KUKA KRL program: PickPlaceTrayTeach.src, PickPlaceTrayTeach.dat

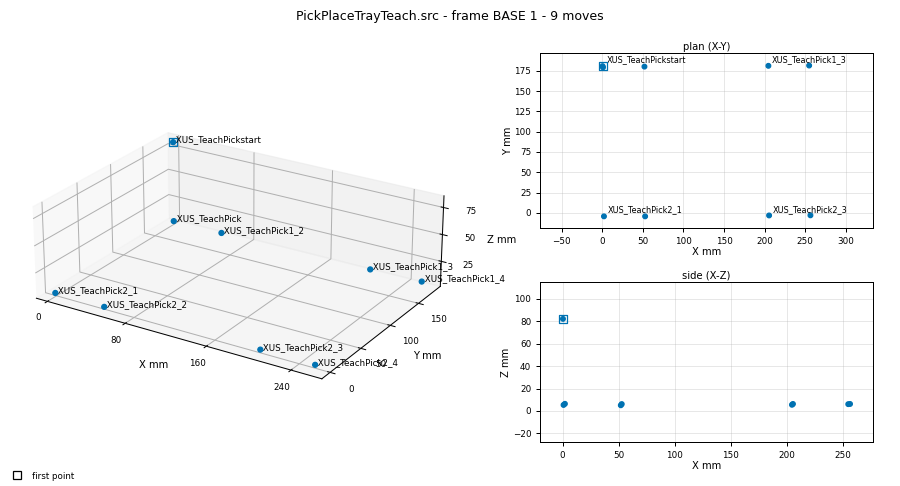
[picture p0: tool path of PickPlaceTrayTeach.src in frame BASE 1, 9 of 139 moves have a stored position in this frame; points joined in program order, loops and branches not executed]
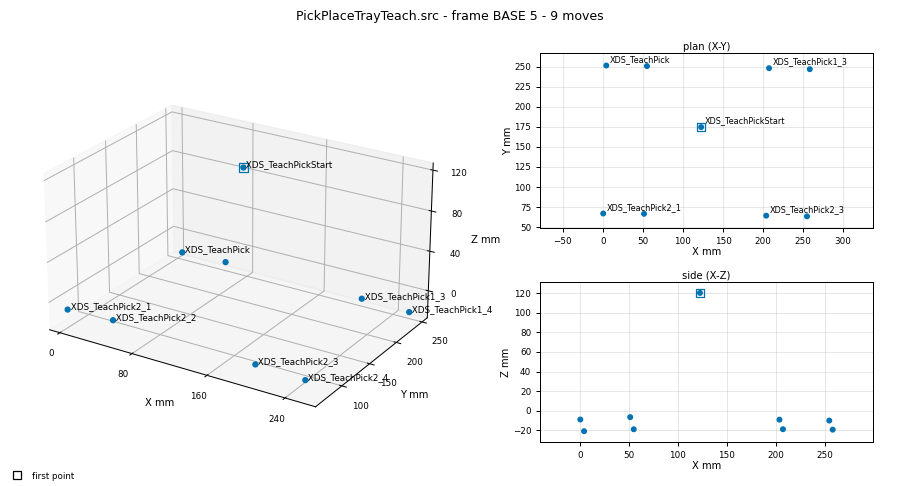
[picture p1: tool path of PickPlaceTrayTeach.src in frame BASE 5, 9 of 139 moves have a stored position in this frame; points joined in program order, loops and branches not executed]
--- PickPlaceTrayTeach.src ---
&ACCESS RVO1
&REL 58
&PARAM DISKPATH = KRC:\R1\Program
DEF PickPlaceTrayTeach()

   ;FOLD INI;%{PE}
      ;FOLD BASISTECH INI
         GLOBAL INTERRUPT DECL 3 WHEN $STOPMESS == TRUE DO IR_STOPM()
         INTERRUPT ON 3
         BAS(#INITMOV, 0)
      ;ENDFOLD (BASISTECH INI)
      ;FOLD USER INI
         ;Make your modifications here
      ;ENDFOLD (USER INI)
      ;ENDFOLD (INI)

            US_Pick[1,1]= XUS_TeachPick
            US_Pick[1,2]= XUS_TeachPick1_2
            US_Pick[1,3]= XUS_TeachPick1_3
            US_Pick[1,4]= XUS_TeachPick1_4
            US_Pick[2,1]= XUS_TeachPick2_1
            US_Pick[2,2]= XUS_TeachPick2_2
            US_Pick[2,3]= XUS_TeachPick2_3
            US_Pick[2,4]= XUS_TeachPick2_4



            DS_Pick[1,1]= XDS_TeachPick
            DS_Pick[1,2]= XDS_TeachPick1_2
            DS_Pick[1,3]= XDS_TeachPick1_3
            DS_Pick[1,4]= XDS_TeachPick1_4
            DS_Pick[2,1]= XDS_TeachPick2_1
            DS_Pick[2,2]= XDS_TeachPick2_2
            DS_Pick[2,3]= XDS_TeachPick2_3
            DS_Pick[2,4]= XDS_TeachPick2_4




            GOTO EndOfModule


        RtoIMM_SeqNumber=1





;move joint 1 to turn robot towards upstacker from home
   ;FOLD SPTP US_A1Turn Vel=100 % PDAT3 Tool[0] Base[0] ;%{PE}
      ;FOLD Parameters ;%{h}
         ;Params IlfProvider=kukaroboter.basistech.inlineforms.movement.spline; Kuka.IsGlobalPoint=False; Kuka.PointName=US_A1Turn; Kuka.BlendingEnabled=False; Kuka.MoveDataPtpName=PDAT3; Kuka.VelocityPtp=100; Kuka.VelocityFieldEnabled=True; Kuka.ColDetectFieldEnabled=True; Kuka.CurrentCDSetIndex=0; Kuka.MovementParameterFieldEnabled=True; IlfCommand=SPTP
      ;ENDFOLD
      SPTP XUS_A1Turn WITH $VEL_AXIS[1] = SVEL_JOINT(100.0), $TOOL = STOOL2(FUS_A1Turn), $BASE = SBASE(FUS_A1Turn.BASE_NO), $IPO_MODE = SIPO_MODE(FUS_A1Turn.IPO_FRAME), $LOAD = SLOAD(FUS_A1Turn.TOOL_NO), $ACC_AXIS[1] = SACC_JOINT(PPDAT3), $APO = SAPO_PTP(PPDAT3), $GEAR_JERK[1] = SGEAR_JERK(PPDAT3), $COLLMON_TOL_PRO[1] = USE_CM_PRO_VALUES(0)
      ;ENDFOLD



;FOLD SPTP US_TeachPickstart Vel=100 % PDAT8 Tool[1]:BlankPick Base[1]:UpStacker ;%{PE}
;FOLD Parameters ;%{h}
;Params IlfProvider=kukaroboter.basistech.inlineforms.movement.spline; Kuka.IsGlobalPoint=False; Kuka.PointName=US_TeachPickstart; Kuka.BlendingEnabled=False; Kuka.MoveDataPtpName=PDAT8; Kuka.VelocityPtp=100; Kuka.VelocityFieldEnabled=True; Kuka.ColDetectFieldEnabled=True; Kuka.CurrentCDSetIndex=0; Kuka.MovementParameterFieldEnabled=True; IlfCommand=SPTP
;ENDFOLD
SPTP XUS_TeachPickstart WITH $VEL_AXIS[1] = SVEL_JOINT(100.0), $TOOL = STOOL2(FUS_TeachPickstart), $BASE = SBASE(FUS_TeachPickstart.BASE_NO), $IPO_MODE = SIPO_MODE(FUS_TeachPickstart.IPO_FRAME), $LOAD = SLOAD(FUS_TeachPickstart.TOOL_NO), $ACC_AXIS[1] = SACC_JOINT(PPDAT8), $APO = SAPO_PTP(PPDAT8), $GEAR_JERK[1] = SGEAR_JERK(PPDAT8), $COLLMON_TOL_PRO[1] = USE_CM_PRO_VALUES(0)
;ENDFOLD

 US_PickApproach[1,1] = US_Pick[1,1]
 US_PickApproach[1,1].Z = US_PickApproach[1,1].Z + 100
 US_PickApproachSlow[1,1].Z = US_PickApproach[1,1].Z - 65
 SLIN US_PickApproach[1,1] with $TOOL=TOOL_DATA[1],$BASE=BASE_DATA[1],$LOAD=LOAD_DATA[1],$VEL.CP = 2
 SLIN US_PickApproachSlow[1,1] with $TOOL=TOOL_DATA[1],$BASE=BASE_DATA[1],$LOAD=LOAD_DATA[1],$VEL.CP = 2
;FOLD SLIN US_TeachPick Vel=1 m/s CPDAT15 Tool[1]:BlankPick Base[1]:UpStacker ;%{PE}
;FOLD Parameters ;%{h}
;Params IlfProvider=kukaroboter.basistech.inlineforms.movement.spline; Kuka.IsGlobalPoint=False; Kuka.PointName=US_TeachPick; Kuka.BlendingEnabled=False; Kuka.MoveDataName=CPDAT15; Kuka.VelocityPath=1; Kuka.VelocityFieldEnabled=True; Kuka.ColDetectFieldEnabled=True; Kuka.CurrentCDSetIndex=0; Kuka.MovementParameterFieldEnabled=True; IlfCommand=SLIN
;ENDFOLD
SLIN XUS_TeachPick WITH $VEL = SVEL_CP(1.0, , LCPDAT15), $TOOL = STOOL2(FUS_TeachPick), $BASE = SBASE(FUS_TeachPick.BASE_NO), $IPO_MODE = SIPO_MODE(FUS_TeachPick.IPO_FRAME), $LOAD = SLOAD(FUS_TeachPick.TOOL_NO), $ACC = SACC_CP(LCPDAT15), $ORI_TYPE = SORI_TYP(LCPDAT15), $APO = SAPO(LCPDAT15), $JERK = SJERK(LCPDAT15), $COLLMON_TOL_PRO[1] = USE_CM_PRO_VALUES(0)
;ENDFOLD
US_Pick[1,1]= XUS_TeachPick
SLIN US_Pick[1,1] with $TOOL=TOOL_DATA[1],$BASE=BASE_DATA[1],$LOAD=LOAD_DATA[1],$VEL.CP = 0.1
SLIN US_PickApproach[1,1] with $TOOL=TOOL_DATA[1],$BASE=BASE_DATA[1],$LOAD=LOAD_DATA[1],$VEL.CP = 2

US_PickApproach[1,2] = US_Pick[1,2]
 US_PickApproach[1,2].Z = US_PickApproach[1,2].Z + 100
 US_PickApproachSlow[1,2].Z = US_PickApproach[1,2].Z - 65
 SLIN US_PickApproach[1,2] with $TOOL=TOOL_DATA[1],$BASE=BASE_DATA[1],$LOAD=LOAD_DATA[1],$VEL.CP = 2
 SLIN US_PickApproachSlow[1,2] with $TOOL=TOOL_DATA[1],$BASE=BASE_DATA[1],$LOAD=LOAD_DATA[1],$VEL.CP = 2
;FOLD SLIN US_TeachPick1_2 Vel=1 m/s CPDAT07 Tool[1]:BlankPick Base[1]:UpStacker ;%{PE}
;FOLD Parameters ;%{h}
;Params IlfProvider=kukaroboter.basistech.inlineforms.movement.spline; Kuka.IsGlobalPoint=False; Kuka.PointName=US_TeachPick1_2; Kuka.BlendingEnabled=False; Kuka.MoveDataName=CPDAT07; Kuka.VelocityPath=1; Kuka.VelocityFieldEnabled=True; Kuka.ColDetectFieldEnabled=True; Kuka.CurrentCDSetIndex=0; Kuka.MovementParameterFieldEnabled=True; IlfCommand=SLIN
;ENDFOLD
SLIN XUS_TeachPick1_2 WITH $VEL = SVEL_CP(1.0, , LCPDAT07), $TOOL = STOOL2(FUS_TeachPick1_2), $BASE = SBASE(FUS_TeachPick1_2.BASE_NO), $IPO_MODE = SIPO_MODE(FUS_TeachPick1_2.IPO_FRAME), $LOAD = SLOAD(FUS_TeachPick1_2.TOOL_NO), $ACC = SACC_CP(LCPDAT07), $ORI_TYPE = SORI_TYP(LCPDAT07), $APO = SAPO(LCPDAT07), $JERK = SJERK(LCPDAT07), $COLLMON_TOL_PRO[1] = USE_CM_PRO_VALUES(0)
;ENDFOLD
US_Pick[1,2]= XUS_TeachPick
SLIN US_Pick[1,2] with $TOOL=TOOL_DATA[1],$BASE=BASE_DATA[1],$LOAD=LOAD_DATA[1],$VEL.CP = 0.1
 SLIN US_PickApproach[1,2] with $TOOL=TOOL_DATA[1],$BASE=BASE_DATA[1],$LOAD=LOAD_DATA[1],$VEL.CP = 2

US_PickApproach[1,3] = US_Pick[1,3]
 US_PickApproach[1,3].Z = US_PickApproach[1,3].Z + 100
 US_PickApproachSlow[1,3].Z = US_PickApproach[1,3].Z - 65
 SLIN US_PickApproach[1,3] with $TOOL=TOOL_DATA[1],$BASE=BASE_DATA[1],$LOAD=LOAD_DATA[1],$VEL.CP = 2
 SLIN US_PickApproachSlow[1,3] with $TOOL=TOOL_DATA[1],$BASE=BASE_DATA[1],$LOAD=LOAD_DATA[1],$VEL.CP = 2
;FOLD SLIN US_TeachPick1_3 Vel=1 m/s CPDAT08 Tool[1]:BlankPick Base[1]:UpStacker ;%{PE}
;FOLD Parameters ;%{h}
;Params IlfProvider=kukaroboter.basistech.inlineforms.movement.spline; Kuka.IsGlobalPoint=False; Kuka.PointName=US_TeachPick1_3; Kuka.BlendingEnabled=False; Kuka.MoveDataName=CPDAT08; Kuka.VelocityPath=1; Kuka.VelocityFieldEnabled=True; Kuka.ColDetectFieldEnabled=True; Kuka.CurrentCDSetIndex=0; Kuka.MovementParameterFieldEnabled=True; IlfCommand=SLIN
;ENDFOLD
SLIN XUS_TeachPick1_3 WITH $VEL = SVEL_CP(1.0, , LCPDAT08), $TOOL = STOOL2(FUS_TeachPick1_3), $BASE = SBASE(FUS_TeachPick1_3.BASE_NO), $IPO_MODE = SIPO_MODE(FUS_TeachPick1_3.IPO_FRAME), $LOAD = SLOAD(FUS_TeachPick1_3.TOOL_NO), $ACC = SACC_CP(LCPDAT08), $ORI_TYPE = SORI_TYP(LCPDAT08), $APO = SAPO(LCPDAT08), $JERK = SJERK(LCPDAT08), $COLLMON_TOL_PRO[1] = USE_CM_PRO_VALUES(0)
;ENDFOLD
US_Pick[1,3]= XUS_TeachPick
SLIN US_Pick[1,3] with $TOOL=TOOL_DATA[1],$BASE=BASE_DATA[1],$LOAD=LOAD_DATA[1],$VEL.CP = 0.1
 SLIN US_PickApproach[1,3] with $TOOL=TOOL_DATA[1],$BASE=BASE_DATA[1],$LOAD=LOAD_DATA[1],$VEL.CP = 2

US_PickApproach[1,4] = US_Pick[1,4]
 US_PickApproach[1,4].Z = US_PickApproach[1,4].Z + 100
 US_PickApproachSlow[1,4].Z = US_PickApproach[1,4].Z - 65
 SLIN US_PickApproach[1,4] with $TOOL=TOOL_DATA[1],$BASE=BASE_DATA[1],$LOAD=LOAD_DATA[1],$VEL.CP = 2
 SLIN US_PickApproachSlow[1,4] with $TOOL=TOOL_DATA[1],$BASE=BASE_DATA[1],$LOAD=LOAD_DATA[1],$VEL.CP = 2
;FOLD SLIN US_TeachPick1_4 Vel=1 m/s CPDAT09 Tool[1]:BlankPick Base[1]:UpStacker ;%{PE}
;FOLD Parameters ;%{h}
;Params IlfProvider=kukaroboter.basistech.inlineforms.movement.spline; Kuka.IsGlobalPoint=False; Kuka.PointName=US_TeachPick1_4; Kuka.BlendingEnabled=False; Kuka.MoveDataName=CPDAT09; Kuka.VelocityPath=1; Kuka.VelocityFieldEnabled=True; Kuka.ColDetectFieldEnabled=True; Kuka.CurrentCDSetIndex=0; Kuka.MovementParameterFieldEnabled=True; IlfCommand=SLIN
;ENDFOLD
SLIN XUS_TeachPick1_4 WITH $VEL = SVEL_CP(1.0, , LCPDAT09), $TOOL = STOOL2(FUS_TeachPick1_4), $BASE = SBASE(FUS_TeachPick1_4.BASE_NO), $IPO_MODE = SIPO_MODE(FUS_TeachPick1_4.IPO_FRAME), $LOAD = SLOAD(FUS_TeachPick1_4.TOOL_NO), $ACC = SACC_CP(LCPDAT09), $ORI_TYPE = SORI_TYP(LCPDAT09), $APO = SAPO(LCPDAT09), $JERK = SJERK(LCPDAT09), $COLLMON_TOL_PRO[1] = USE_CM_PRO_VALUES(0)
;ENDFOLD
US_Pick[1,4]= XUS_TeachPick
SLIN US_Pick[1,4] with $TOOL=TOOL_DATA[1],$BASE=BASE_DATA[1],$LOAD=LOAD_DATA[1],$VEL.CP = 0.1
 SLIN US_PickApproach[1,4] with $TOOL=TOOL_DATA[1],$BASE=BASE_DATA[1],$LOAD=LOAD_DATA[1],$VEL.CP = 2

US_PickApproach[2,1] = US_Pick[2,1]
 US_PickApproach[2,1].Z = US_PickApproach[2,1].Z + 100
 US_PickApproachSlow[2,1].Z = US_PickApproach[2,1].Z - 65
 SLIN US_PickApproach[2,1] with $TOOL=TOOL_DATA[1],$BASE=BASE_DATA[1],$LOAD=LOAD_DATA[1],$VEL.CP = 2
 SLIN US_PickApproachSlow[2,1] with $TOOL=TOOL_DATA[1],$BASE=BASE_DATA[1],$LOAD=LOAD_DATA[1],$VEL.CP = 2
;FOLD SLIN US_TeachPick2_1 Vel=1 m/s CPDAT11 Tool[1]:BlankPick Base[1]:UpStacker ;%{PE}
;FOLD Parameters ;%{h}
;Params IlfProvider=kukaroboter.basistech.inlineforms.movement.spline; Kuka.IsGlobalPoint=False; Kuka.PointName=US_TeachPick2_1; Kuka.BlendingEnabled=False; Kuka.MoveDataName=CPDAT11; Kuka.VelocityPath=1; Kuka.VelocityFieldEnabled=True; Kuka.ColDetectFieldEnabled=True; Kuka.CurrentCDSetIndex=0; Kuka.MovementParameterFieldEnabled=True; IlfCommand=SLIN
;ENDFOLD
SLIN XUS_TeachPick2_1 WITH $VEL = SVEL_CP(1.0, , LCPDAT11), $TOOL = STOOL2(FUS_TeachPick2_1), $BASE = SBASE(FUS_TeachPick2_1.BASE_NO), $IPO_MODE = SIPO_MODE(FUS_TeachPick2_1.IPO_FRAME), $LOAD = SLOAD(FUS_TeachPick2_1.TOOL_NO), $ACC = SACC_CP(LCPDAT11), $ORI_TYPE = SORI_TYP(LCPDAT11), $APO = SAPO(LCPDAT11), $JERK = SJERK(LCPDAT11), $COLLMON_TOL_PRO[1] = USE_CM_PRO_VALUES(0)
;ENDFOLD
US_Pick[2,1]= XUS_TeachPick
SLIN US_Pick[2,1] with $TOOL=TOOL_DATA[1],$BASE=BASE_DATA[1],$LOAD=LOAD_DATA[1],$VEL.CP = 0.1
 SLIN US_PickApproach[2,1] with $TOOL=TOOL_DATA[1],$BASE=BASE_DATA[1],$LOAD=LOAD_DATA[1],$VEL.CP = 2

US_PickApproach[2,2] = US_Pick[2,2]
 US_PickApproach[2,2].Z = US_PickApproach[2,2].Z + 100
 US_PickApproachSlow[2,2].Z = US_PickApproach[2,2].Z - 65
 SLIN US_PickApproach[2,2] with $TOOL=TOOL_DATA[1],$BASE=BASE_DATA[1],$LOAD=LOAD_DATA[1],$VEL.CP = 2
 SLIN US_PickApproachSlow[2,2] with $TOOL=TOOL_DATA[1],$BASE=BASE_DATA[1],$LOAD=LOAD_DATA[1],$VEL.CP = 2
;FOLD SLIN US_TeachPick2_2 Vel=1 m/s CPDAT12 Tool[1]:BlankPick Base[1]:UpStacker ;%{PE}
;FOLD Parameters ;%{h}
;Params IlfProvider=kukaroboter.basistech.inlineforms.movement.spline; Kuka.IsGlobalPoint=False; Kuka.PointName=US_TeachPick2_2; Kuka.BlendingEnabled=False; Kuka.MoveDataName=CPDAT12; Kuka.VelocityPath=1; Kuka.VelocityFieldEnabled=True; Kuka.ColDetectFieldEnabled=True; Kuka.CurrentCDSetIndex=0; Kuka.MovementParameterFieldEnabled=True; IlfCommand=SLIN
;ENDFOLD
SLIN XUS_TeachPick2_2 WITH $VEL = SVEL_CP(1.0, , LCPDAT12), $TOOL = STOOL2(FUS_TeachPick2_2), $BASE = SBASE(FUS_TeachPick2_2.BASE_NO), $IPO_MODE = SIPO_MODE(FUS_TeachPick2_2.IPO_FRAME), $LOAD = SLOAD(FUS_TeachPick2_2.TOOL_NO), $ACC = SACC_CP(LCPDAT12), $ORI_TYPE = SORI_TYP(LCPDAT12), $APO = SAPO(LCPDAT12), $JERK = SJERK(LCPDAT12), $COLLMON_TOL_PRO[1] = USE_CM_PRO_VALUES(0)
;ENDFOLD
US_Pick[2,2]= XUS_TeachPick
SLIN US_Pick[2,2] with $TOOL=TOOL_DATA[1],$BASE=BASE_DATA[1],$LOAD=LOAD_DATA[1],$VEL.CP = 0.1
SLIN US_PickApproach[2,2] with $TOOL=TOOL_DATA[1],$BASE=BASE_DATA[1],$LOAD=LOAD_DATA[1],$VEL.CP = 2

US_PickApproach[2,3] = US_Pick[2,3]
 US_PickApproach[2,3].Z = US_PickApproach[2,3].Z + 100
 US_PickApproachSlow[2,3].Z = US_PickApproach[2,3].Z - 65
 SLIN US_PickApproach[2,3] with $TOOL=TOOL_DATA[1],$BASE=BASE_DATA[1],$LOAD=LOAD_DATA[1],$VEL.CP = 2
 SLIN US_PickApproachSlow[2,3] with $TOOL=TOOL_DATA[1],$BASE=BASE_DATA[1],$LOAD=LOAD_DATA[1],$VEL.CP = 2
;FOLD SLIN US_TeachPick2_3 Vel=1 m/s CPDAT13 Tool[1]:BlankPick Base[1]:UpStacker ;%{PE}
;FOLD Parameters ;%{h}
;Params IlfProvider=kukaroboter.basistech.inlineforms.movement.spline; Kuka.IsGlobalPoint=False; Kuka.PointName=US_TeachPick2_3; Kuka.BlendingEnabled=False; Kuka.MoveDataName=CPDAT13; Kuka.VelocityPath=1; Kuka.VelocityFieldEnabled=True; Kuka.ColDetectFieldEnabled=True; Kuka.CurrentCDSetIndex=0; Kuka.MovementParameterFieldEnabled=True; IlfCommand=SLIN
;ENDFOLD
SLIN XUS_TeachPick2_3 WITH $VEL = SVEL_CP(1.0, , LCPDAT13), $TOOL = STOOL2(FUS_TeachPick2_3), $BASE = SBASE(FUS_TeachPick2_3.BASE_NO), $IPO_MODE = SIPO_MODE(FUS_TeachPick2_3.IPO_FRAME), $LOAD = SLOAD(FUS_TeachPick2_3.TOOL_NO), $ACC = SACC_CP(LCPDAT13), $ORI_TYPE = SORI_TYP(LCPDAT13), $APO = SAPO(LCPDAT13), $JERK = SJERK(LCPDAT13), $COLLMON_TOL_PRO[1] = USE_CM_PRO_VALUES(0)
;ENDFOLD
US_Pick[2,3]= XUS_TeachPick
SLIN US_Pick[2,3] with $TOOL=TOOL_DATA[1],$BASE=BASE_DATA[1],$LOAD=LOAD_DATA[1],$VEL.CP = 0.1
SLIN US_PickApproach[2,3] with $TOOL=TOOL_DATA[1],$BASE=BASE_DATA[1],$LOAD=LOAD_DATA[1],$VEL.CP = 2

US_PickApproach[2,4] = US_Pick[2,4]
 US_PickApproach[2,4].Z = US_PickApproach[2,4].Z + 100
 US_PickApproachSlow[2,4].Z = US_PickApproach[2,4].Z - 65
 SLIN US_PickApproach[2,4] with $TOOL=TOOL_DATA[1],$BASE=BASE_DATA[1],$LOAD=LOAD_DATA[1],$VEL.CP = 2
 SLIN US_PickApproachSlow[2,4] with $TOOL=TOOL_DATA[1],$BASE=BASE_DATA[1],$LOAD=LOAD_DATA[1],$VEL.CP = 2
;FOLD SLIN US_TeachPick2_4 Vel=1 m/s CPDAT14 Tool[1]:BlankPick Base[1]:UpStacker ;%{PE}
;FOLD Parameters ;%{h}
;Params IlfProvider=kukaroboter.basistech.inlineforms.movement.spline; Kuka.IsGlobalPoint=False; Kuka.PointName=US_TeachPick2_4; Kuka.BlendingEnabled=False; Kuka.MoveDataName=CPDAT14; Kuka.VelocityPath=1; Kuka.VelocityFieldEnabled=True; Kuka.ColDetectFieldEnabled=True; Kuka.CurrentCDSetIndex=0; Kuka.MovementParameterFieldEnabled=True; IlfCommand=SLIN
;ENDFOLD
SLIN XUS_TeachPick2_4 WITH $VEL = SVEL_CP(1.0, , LCPDAT14), $TOOL = STOOL2(FUS_TeachPick2_4), $BASE = SBASE(FUS_TeachPick2_4.BASE_NO), $IPO_MODE = SIPO_MODE(FUS_TeachPick2_4.IPO_FRAME), $LOAD = SLOAD(FUS_TeachPick2_4.TOOL_NO), $ACC = SACC_CP(LCPDAT14), $ORI_TYPE = SORI_TYP(LCPDAT14), $APO = SAPO(LCPDAT14), $JERK = SJERK(LCPDAT14), $COLLMON_TOL_PRO[1] = USE_CM_PRO_VALUES(0)
;ENDFOLD
US_Pick[2,4]= XUS_TeachPick
SLIN US_Pick[2,4] with $TOOL=TOOL_DATA[1],$BASE=BASE_DATA[1],$LOAD=LOAD_DATA[1],$VEL.CP = 0.1
SLIN US_PickApproach[2,4] with $TOOL=TOOL_DATA[1],$BASE=BASE_DATA[1],$LOAD=LOAD_DATA[1],$VEL.CP = 2























;FOLD SPTP DS_TeachPickStart Vel=100 % PDAT12 Tool[2]:FinishedPlace Base[5]:DownStacker ;%{PE}
;FOLD Parameters ;%{h}
;Params IlfProvider=kukaroboter.basistech.inlineforms.movement.spline; Kuka.IsGlobalPoint=False; Kuka.PointName=DS_TeachPickStart; Kuka.BlendingEnabled=False; Kuka.MoveDataPtpName=PDAT12; Kuka.VelocityPtp=100; Kuka.VelocityFieldEnabled=True; Kuka.ColDetectFieldEnabled=True; Kuka.CurrentCDSetIndex=0; Kuka.MovementParameterFieldEnabled=True; IlfCommand=SPTP
;ENDFOLD
SPTP XDS_TeachPickStart WITH $VEL_AXIS[1] = SVEL_JOINT(100.0), $TOOL = STOOL2(FDS_TeachPickStart), $BASE = SBASE(FDS_TeachPickStart.BASE_NO), $IPO_MODE = SIPO_MODE(FDS_TeachPickStart.IPO_FRAME), $LOAD = SLOAD(FDS_TeachPickStart.TOOL_NO), $ACC_AXIS[1] = SACC_JOINT(PPDAT12), $APO = SAPO_PTP(PPDAT12), $GEAR_JERK[1] = SGEAR_JERK(PPDAT12), $COLLMON_TOL_PRO[1] = USE_CM_PRO_VALUES(0)
;ENDFOLD

 DS_PickApproach[1,1] = DS_Pick[1,1]
 DS_PickApproach[1,1].Z = DS_PickApproach[1,1].Z + 100
 DS_PickApproachSlow[1,1].Z = DS_PickApproach[1,1].Z - 65
 SLIN DS_PickApproach[1,1] with $TOOL=TOOL_DATA[1],$BASE=BASE_DATA[1],$LOAD=LOAD_DATA[1],$VEL.CP = 2
 SLIN DS_PickApproachSlow[1,1] with $TOOL=TOOL_DATA[1],$BASE=BASE_DATA[1],$LOAD=LOAD_DATA[1],$VEL.CP = 2
;FOLD SLIN DS_TeachPick Vel=1 m/s CPDAT21 Tool[2]:FinishedPlace Base[5]:DownStacker ;%{PE}
;FOLD Parameters ;%{h}
;Params IlfProvider=kukaroboter.basistech.inlineforms.movement.spline; Kuka.IsGlobalPoint=False; Kuka.PointName=DS_TeachPick; Kuka.BlendingEnabled=False; Kuka.MoveDataName=CPDAT21; Kuka.VelocityPath=1; Kuka.VelocityFieldEnabled=True; Kuka.ColDetectFieldEnabled=True; Kuka.CurrentCDSetIndex=0; Kuka.MovementParameterFieldEnabled=True; IlfCommand=SLIN
;ENDFOLD
SLIN XDS_TeachPick WITH $VEL = SVEL_CP(1.0, , LCPDAT21), $TOOL = STOOL2(FDS_TeachPick), $BASE = SBASE(FDS_TeachPick.BASE_NO), $IPO_MODE = SIPO_MODE(FDS_TeachPick.IPO_FRAME), $LOAD = SLOAD(FDS_TeachPick.TOOL_NO), $ACC = SACC_CP(LCPDAT21), $ORI_TYPE = SORI_TYP(LCPDAT21), $APO = SAPO(LCPDAT21), $JERK = SJERK(LCPDAT21), $COLLMON_TOL_PRO[1] = USE_CM_PRO_VALUES(0)
;ENDFOLD
DS_Pick[1,1]= XUS_TeachPick
SLIN DS_Pick[1,1] with $TOOL=TOOL_DATA[1],$BASE=BASE_DATA[1],$LOAD=LOAD_DATA[1],$VEL.CP = 0.1
SLIN DS_PickApproach[1,1] with $TOOL=TOOL_DATA[1],$BASE=BASE_DATA[1],$LOAD=LOAD_DATA[1],$VEL.CP = 2


DS_PickApproach[1,2] = DS_Pick[1,2]
 DS_PickApproach[1,2].Z = DS_PickApproach[1,2].Z + 100
 DS_PickApproachSlow[1,2].Z = DS_PickApproach[1,2].Z - 65
 SLIN DS_PickApproach[1,2] with $TOOL=TOOL_DATA[1],$BASE=BASE_DATA[1],$LOAD=LOAD_DATA[1],$VEL.CP = 2
 SLIN DS_PickApproachSlow[1,2] with $TOOL=TOOL_DATA[1],$BASE=BASE_DATA[1],$LOAD=LOAD_DATA[1],$VEL.CP = 2
;FOLD SLIN DS_TeachPick1_2 Vel=1 m/s CPDAT19 Tool[2]:FinishedPlace Base[5]:DownStacker ;%{PE}
;FOLD Parameters ;%{h}
;Params IlfProvider=kukaroboter.basistech.inlineforms.movement.spline; Kuka.IsGlobalPoint=False; Kuka.PointName=DS_TeachPick1_2; Kuka.BlendingEnabled=False; Kuka.MoveDataName=CPDAT19; Kuka.VelocityPath=1; Kuka.VelocityFieldEnabled=True; Kuka.ColDetectFieldEnabled=True; Kuka.CurrentCDSetIndex=0; Kuka.MovementParameterFieldEnabled=True; IlfCommand=SLIN
;ENDFOLD
SLIN XDS_TeachPick1_2 WITH $VEL = SVEL_CP(1.0, , LCPDAT19), $TOOL = STOOL2(FDS_TeachPick1_2), $BASE = SBASE(FDS_TeachPick1_2.BASE_NO), $IPO_MODE = SIPO_MODE(FDS_TeachPick1_2.IPO_FRAME), $LOAD = SLOAD(FDS_TeachPick1_2.TOOL_NO), $ACC = SACC_CP(LCPDAT19), $ORI_TYPE = SORI_TYP(LCPDAT19), $APO = SAPO(LCPDAT19), $JERK = SJERK(LCPDAT19), $COLLMON_TOL_PRO[1] = USE_CM_PRO_VALUES(0)
;ENDFOLD
DS_Pick[1,2]= XUS_TeachPick
SLIN DS_Pick[1,2] with $TOOL=TOOL_DATA[1],$BASE=BASE_DATA[1],$LOAD=LOAD_DATA[1],$VEL.CP = 0.1
 SLIN DS_PickApproach[1,2] with $TOOL=TOOL_DATA[1],$BASE=BASE_DATA[1],$LOAD=LOAD_DATA[1],$VEL.CP = 2


DS_PickApproach[1,3] = DS_Pick[1,3]
 DS_PickApproach[1,3].Z = DS_PickApproach[1,3].Z + 100
 DS_PickApproachSlow[1,3].Z = DS_PickApproach[1,3].Z - 65
 SLIN DS_PickApproach[1,3] with $TOOL=TOOL_DATA[1],$BASE=BASE_DATA[1],$LOAD=LOAD_DATA[1],$VEL.CP = 2
 SLIN DS_PickApproachSlow[1,3] with $TOOL=TOOL_DATA[1],$BASE=BASE_DATA[1],$LOAD=LOAD_DATA[1],$VEL.CP = 2
;FOLD SLIN DS_TeachPick1_3 Vel=1 m/s CPDAT18 Tool[2]:FinishedPlace Base[5]:DownStacker ;%{PE}
;FOLD Parameters ;%{h}
;Params IlfProvider=kukaroboter.basistech.inlineforms.movement.spline; Kuka.IsGlobalPoint=False; Kuka.PointName=DS_TeachPick1_3; Kuka.BlendingEnabled=False; Kuka.MoveDataName=CPDAT18; Kuka.VelocityPath=1; Kuka.VelocityFieldEnabled=True; Kuka.ColDetectFieldEnabled=True; Kuka.CurrentCDSetIndex=0; Kuka.MovementParameterFieldEnabled=True; IlfCommand=SLIN
;ENDFOLD
SLIN XDS_TeachPick1_3 WITH $VEL = SVEL_CP(1.0, , LCPDAT18), $TOOL = STOOL2(FDS_TeachPick1_3), $BASE = SBASE(FDS_TeachPick1_3.BASE_NO), $IPO_MODE = SIPO_MODE(FDS_TeachPick1_3.IPO_FRAME), $LOAD = SLOAD(FDS_TeachPick1_3.TOOL_NO), $ACC = SACC_CP(LCPDAT18), $ORI_TYPE = SORI_TYP(LCPDAT18), $APO = SAPO(LCPDAT18), $JERK = SJERK(LCPDAT18), $COLLMON_TOL_PRO[1] = USE_CM_PRO_VALUES(0)
;ENDFOLD
DS_Pick[1,3]= XUS_TeachPick
SLIN DS_Pick[1,3] with $TOOL=TOOL_DATA[1],$BASE=BASE_DATA[1],$LOAD=LOAD_DATA[1],$VEL.CP = 0.1
 SLIN DS_PickApproach[1,3] with $TOOL=TOOL_DATA[1],$BASE=BASE_DATA[1],$LOAD=LOAD_DATA[1],$VEL.CP = 2


DS_PickApproach[1,4] = DS_Pick[1,4]
 DS_PickApproach[1,4].Z = DS_PickApproach[1,4].Z + 100
 DS_PickApproachSlow[1,4].Z = DS_PickApproach[1,4].Z - 65
 SLIN DS_PickApproach[1,4] with $TOOL=TOOL_DATA[1],$BASE=BASE_DATA[1],$LOAD=LOAD_DATA[1],$VEL.CP = 2
 SLIN DS_PickApproachSlow[1,4] with $TOOL=TOOL_DATA[1],$BASE=BASE_DATA[1],$LOAD=LOAD_DATA[1],$VEL.CP = 2
;FOLD SLIN DS_TeachPick1_4 Vel=1 m/s CPDAT20 Tool[2]:FinishedPlace Base[5]:DownStacker ;%{PE}
;FOLD Parameters ;%{h}
;Params IlfProvider=kukaroboter.basistech.inlineforms.movement.spline; Kuka.IsGlobalPoint=False; Kuka.PointName=DS_TeachPick1_4; Kuka.BlendingEnabled=False; Kuka.MoveDataName=CPDAT20; Kuka.VelocityPath=1; Kuka.VelocityFieldEnabled=True; Kuka.ColDetectFieldEnabled=True; Kuka.CurrentCDSetIndex=0; Kuka.MovementParameterFieldEnabled=True; IlfCommand=SLIN
;ENDFOLD
SLIN XDS_TeachPick1_4 WITH $VEL = SVEL_CP(1.0, , LCPDAT20), $TOOL = STOOL2(FDS_TeachPick1_4), $BASE = SBASE(FDS_TeachPick1_4.BASE_NO), $IPO_MODE = SIPO_MODE(FDS_TeachPick1_4.IPO_FRAME), $LOAD = SLOAD(FDS_TeachPick1_4.TOOL_NO), $ACC = SACC_CP(LCPDAT20), $ORI_TYPE = SORI_TYP(LCPDAT20), $APO = SAPO(LCPDAT20), $JERK = SJERK(LCPDAT20), $COLLMON_TOL_PRO[1] = USE_CM_PRO_VALUES(0)
;ENDFOLD
DS_Pick[1,4]= XUS_TeachPick
SLIN DS_Pick[1,4] with $TOOL=TOOL_DATA[1],$BASE=BASE_DATA[1],$LOAD=LOAD_DATA[1],$VEL.CP = 0.1
 SLIN DS_PickApproach[1,4] with $TOOL=TOOL_DATA[1],$BASE=BASE_DATA[1],$LOAD=LOAD_DATA[1],$VEL.CP = 2


DS_PickApproach[2,1] = DS_Pick[2,1]
 DS_PickApproach[2,1].Z = DS_PickApproach[2,1].Z + 100
 DS_PickApproachSlow[2,1].Z = DS_PickApproach[2,1].Z - 65
 SLIN DS_PickApproach[2,1] with $TOOL=TOOL_DATA[1],$BASE=BASE_DATA[1],$LOAD=LOAD_DATA[1],$VEL.CP = 2
 SLIN DS_PickApproachSlow[2,1] with $TOOL=TOOL_DATA[1],$BASE=BASE_DATA[1],$LOAD=LOAD_DATA[1],$VEL.CP = 2
;FOLD SLIN DS_TeachPick2_1 Vel=1 m/s CPDAT22 Tool[2]:FinishedPlace Base[5]:DownStacker ;%{PE}
;FOLD Parameters ;%{h}
;Params IlfProvider=kukaroboter.basistech.inlineforms.movement.spline; Kuka.IsGlobalPoint=False; Kuka.PointName=DS_TeachPick2_1; Kuka.BlendingEnabled=False; Kuka.MoveDataName=CPDAT22; Kuka.VelocityPath=1; Kuka.VelocityFieldEnabled=True; Kuka.ColDetectFieldEnabled=True; Kuka.CurrentCDSetIndex=0; Kuka.MovementParameterFieldEnabled=True; IlfCommand=SLIN
;ENDFOLD
SLIN XDS_TeachPick2_1 WITH $VEL = SVEL_CP(1.0, , LCPDAT22), $TOOL = STOOL2(FDS_TeachPick2_1), $BASE = SBASE(FDS_TeachPick2_1.BASE_NO), $IPO_MODE = SIPO_MODE(FDS_TeachPick2_1.IPO_FRAME), $LOAD = SLOAD(FDS_TeachPick2_1.TOOL_NO), $ACC = SACC_CP(LCPDAT22), $ORI_TYPE = SORI_TYP(LCPDAT22), $APO = SAPO(LCPDAT22), $JERK = SJERK(LCPDAT22), $COLLMON_TOL_PRO[1] = USE_CM_PRO_VALUES(0)
;ENDFOLD
DS_Pick[2,1]= XUS_TeachPick
SLIN DS_Pick[2,1] with $TOOL=TOOL_DATA[1],$BASE=BASE_DATA[1],$LOAD=LOAD_DATA[1],$VEL.CP = 0.1
 SLIN DS_PickApproach[2,1] with $TOOL=TOOL_DATA[1],$BASE=BASE_DATA[1],$LOAD=LOAD_DATA[1],$VEL.CP = 2


DS_PickApproach[2,2] = DS_Pick[2,2]
 DS_PickApproach[2,2].Z = DS_PickApproach[2,2].Z + 100
 DS_PickApproachSlow[2,2].Z = DS_PickApproach[2,2].Z - 65
 SLIN DS_PickApproach[2,2] with $TOOL=TOOL_DATA[1],$BASE=BASE_DATA[1],$LOAD=LOAD_DATA[1],$VEL.CP = 2
 SLIN DS_PickApproachSlow[2,2] with $TOOL=TOOL_DATA[1],$BASE=BASE_DATA[1],$LOAD=LOAD_DATA[1],$VEL.CP = 2
;FOLD SLIN DS_TeachPick2_2 Vel=1 m/s CPDAT23 Tool[2]:FinishedPlace Base[5]:DownStacker ;%{PE}
;FOLD Parameters ;%{h}
;Params IlfProvider=kukaroboter.basistech.inlineforms.movement.spline; Kuka.IsGlobalPoint=False; Kuka.PointName=DS_TeachPick2_2; Kuka.BlendingEnabled=False; Kuka.MoveDataName=CPDAT23; Kuka.VelocityPath=1; Kuka.VelocityFieldEnabled=True; Kuka.ColDetectFieldEnabled=True; Kuka.CurrentCDSetIndex=0; Kuka.MovementParameterFieldEnabled=True; IlfCommand=SLIN
;ENDFOLD
SLIN XDS_TeachPick2_2 WITH $VEL = SVEL_CP(1.0, , LCPDAT23), $TOOL = STOOL2(FDS_TeachPick2_2), $BASE = SBASE(FDS_TeachPick2_2.BASE_NO), $IPO_MODE = SIPO_MODE(FDS_TeachPick2_2.IPO_FRAME), $LOAD = SLOAD(FDS_TeachPick2_2.TOOL_NO), $ACC = SACC_CP(LCPDAT23), $ORI_TYPE = SORI_TYP(LCPDAT23), $APO = SAPO(LCPDAT23), $JERK = SJERK(LCPDAT23), $COLLMON_TOL_PRO[1] = USE_CM_PRO_VALUES(0)
;ENDFOLD
DS_Pick[2,2]= XUS_TeachPick
SLIN DS_Pick[2,2] with $TOOL=TOOL_DATA[1],$BASE=BASE_DATA[1],$LOAD=LOAD_DATA[1],$VEL.CP = 0.1
SLIN DS_PickApproach[2,2] with $TOOL=TOOL_DATA[1],$BASE=BASE_DATA[1],$LOAD=LOAD_DATA[1],$VEL.CP = 2


DS_PickApproach[2,3] = DS_Pick[2,3]
 DS_PickApproach[2,3].Z = DS_PickApproach[2,3].Z + 100
 DS_PickApproachSlow[2,3].Z = DS_PickApproach[2,3].Z - 65
 SLIN DS_PickApproach[2,3] with $TOOL=TOOL_DATA[1],$BASE=BASE_DATA[1],$LOAD=LOAD_DATA[1],$VEL.CP = 2
 SLIN DS_PickApproachSlow[2,3] with $TOOL=TOOL_DATA[1],$BASE=BASE_DATA[1],$LOAD=LOAD_DATA[1],$VEL.CP = 2
;FOLD SLIN DS_TeachPick2_3 Vel=1 m/s CPDAT24 Tool[2]:FinishedPlace Base[5]:DownStacker ;%{PE}
;FOLD Parameters ;%{h}
;Params IlfProvider=kukaroboter.basistech.inlineforms.movement.spline; Kuka.IsGlobalPoint=False; Kuka.PointName=DS_TeachPick2_3; Kuka.BlendingEnabled=False; Kuka.MoveDataName=CPDAT24; Kuka.VelocityPath=1; Kuka.VelocityFieldEnabled=True; Kuka.ColDetectFieldEnabled=True; Kuka.CurrentCDSetIndex=0; Kuka.MovementParameterFieldEnabled=True; IlfCommand=SLIN
;ENDFOLD
SLIN XDS_TeachPick2_3 WITH $VEL = SVEL_CP(1.0, , LCPDAT24), $TOOL = STOOL2(FDS_TeachPick2_3), $BASE = SBASE(FDS_TeachPick2_3.BASE_NO), $IPO_MODE = SIPO_MODE(FDS_TeachPick2_3.IPO_FRAME), $LOAD = SLOAD(FDS_TeachPick2_3.TOOL_NO), $ACC = SACC_CP(LCPDAT24), $ORI_TYPE = SORI_TYP(LCPDAT24), $APO = SAPO(LCPDAT24), $JERK = SJERK(LCPDAT24), $COLLMON_TOL_PRO[1] = USE_CM_PRO_VALUES(0)
;ENDFOLD
DS_Pick[2,3]= XUS_TeachPick
SLIN DS_Pick[2,3] with $TOOL=TOOL_DATA[1],$BASE=BASE_DATA[1],$LOAD=LOAD_DATA[1],$VEL.CP = 0.1
SLIN DS_PickApproach[2,3] with $TOOL=TOOL_DATA[1],$BASE=BASE_DATA[1],$LOAD=LOAD_DATA[1],$VEL.CP = 2


DS_PickApproach[2,4] = DS_Pick[2,4]
 DS_PickApproach[2,4].Z = DS_PickApproach[2,4].Z + 100
 DS_PickApproachSlow[2,4].Z = DS_PickApproach[2,4].Z - 65
 SLIN DS_PickApproach[2,4] with $TOOL=TOOL_DATA[1],$BASE=BASE_DATA[1],$LOAD=LOAD_DATA[1],$VEL.CP = 2
 SLIN DS_PickApproachSlow[2,4] with $TOOL=TOOL_DATA[1],$BASE=BASE_DATA[1],$LOAD=LOAD_DATA[1],$VEL.CP = 2
;FOLD SLIN DS_TeachPick2_4 Vel=1 m/s CPDAT25 Tool[2]:FinishedPlace Base[5]:DownStacker ;%{PE}
;FOLD Parameters ;%{h}
;Params IlfProvider=kukaroboter.basistech.inlineforms.movement.spline; Kuka.IsGlobalPoint=False; Kuka.PointName=DS_TeachPick2_4; Kuka.BlendingEnabled=False; Kuka.MoveDataName=CPDAT25; Kuka.VelocityPath=1; Kuka.VelocityFieldEnabled=True; Kuka.ColDetectFieldEnabled=True; Kuka.CurrentCDSetIndex=0; Kuka.MovementParameterFieldEnabled=True; IlfCommand=SLIN
;ENDFOLD
SLIN XDS_TeachPick2_4 WITH $VEL = SVEL_CP(1.0, , LCPDAT25), $TOOL = STOOL2(FDS_TeachPick2_4), $BASE = SBASE(FDS_TeachPick2_4.BASE_NO), $IPO_MODE = SIPO_MODE(FDS_TeachPick2_4.IPO_FRAME), $LOAD = SLOAD(FDS_TeachPick2_4.TOOL_NO), $ACC = SACC_CP(LCPDAT25), $ORI_TYPE = SORI_TYP(LCPDAT25), $APO = SAPO(LCPDAT25), $JERK = SJERK(LCPDAT25), $COLLMON_TOL_PRO[1] = USE_CM_PRO_VALUES(0)
;ENDFOLD
DS_Pick[2,4]= XUS_TeachPick
SLIN DS_Pick[2,4] with $TOOL=TOOL_DATA[1],$BASE=BASE_DATA[1],$LOAD=LOAD_DATA[1],$VEL.CP = 0.1
SLIN DS_PickApproach[2,4] with $TOOL=TOOL_DATA[1],$BASE=BASE_DATA[1],$LOAD=LOAD_DATA[1],$VEL.CP = 2







;Clear vacuum cups outputs
RtoPLC_BlankCupAVac=False
RtoPLC_BlankCupBVac=False
RtoPLC_BlankCupABlow=False
RtoPLC_BlankCupBBlow=False







halt


 ;move tooling to row and column approach position for pick, then slowy move into the pick position
            US_PickApproach[1,1] = US_Pick[1,1]
            US_PickApproach[1,1].Z = US_PickApproach[1,1].Z + 100
            US_PickApproachSlow[1,1].Z = US_PickApproach[1,1].Z - 65
            US_Pick1[1,1]= US_Pick[1,1]
            US_Pick2[1,1]= US_Pick[1,1]
            US_Pick3[1,1]= US_Pick[1,1]
            US_Pick1[1,1].X = US_Pick[1,1].X + 0.009187222
            US_Pick1[1,1].Y = US_Pick[1,1].Y  -0.805848
            US_Pick1[1,1].Z = US_Pick[1,1].Z + 0.81393918
            US_Pick1[1,1].A = US_Pick[1,1].A + 0.00272370000000421
            US_Pick1[1,1].B = US_Pick[1,1].B -0.999994156
            US_Pick1[1,1].C = US_Pick[1,1].C -0.00344900000001758
            US_Pick2[1,1].X = US_Pick[1,1].X -1.830273332
            US_Pick2[1,1].Y = US_Pick[1,1].Y  + 0.118088
            US_Pick2[1,1].Z = US_Pick[1,1].Z + 0.22346
            US_Pick2[1,1].A = US_Pick[1,1].A + 0.00272370000000421
            US_Pick2[1,1].B = US_Pick[1,1].B -0.999994156
            US_Pick2[1,1].C = US_Pick[1,1].C -0.00344900000001758
            US_Pick3[1,1].X = US_Pick[1,1].X + 0.764676273
            US_Pick3[1,1].Y = US_Pick[1,1].Y  -1.519576
            US_Pick3[1,1].Z = US_Pick[1,1].Z -0.17324344
            US_Pick3[1,1].A = US_Pick[1,1].A + 0.00272370000000421
            US_Pick3[1,1].B = US_Pick[1,1].B -0.999990132
            US_Pick3[1,1].C = US_Pick[1,1].C -0.00344900000001758
 RtoPLC_BlankCupAVac=False
RtoPLC_BlankCupBVac=False
RtoPLC_BlankCupABlow=False
RtoPLC_BlankCupBBlow=False
 SPTP US_PickApproach[1,1] with $TOOL=TOOL_DATA[1],$BASE=BASE_DATA[1],$LOAD=LOAD_DATA[1],$VEL.CP = 2
 SLIN US_PickApproachSlow[1,1] with $TOOL=TOOL_DATA[1],$BASE=BASE_DATA[1],$LOAD=LOAD_DATA[1],$VEL.CP = 2
 SLIN US_Pick1[1,1] with $TOOL=TOOL_DATA[1],$BASE=BASE_DATA[1],$LOAD=LOAD_DATA[1],$VEL.CP = .01
 SLIN US_Pick2[1,1] with $TOOL=TOOL_DATA[1],$BASE=BASE_DATA[1],$LOAD=LOAD_DATA[1],$VEL.CP = 1
 SLIN US_Pick3[1,1] with $TOOL=TOOL_DATA[1],$BASE=BASE_DATA[1],$LOAD=LOAD_DATA[1],$VEL.CP = 1
 SLIN US_Pick[1,1] with $TOOL=TOOL_DATA[1],$BASE=BASE_DATA[1],$LOAD=LOAD_DATA[1],$VEL.CP = 1

RtoPLC_BlankCupAVac=True
RtoPLC_BlankCupBVac=True
SLIN US_PickApproachSlow[1,1] with $TOOL=TOOL_DATA[1],$BASE=BASE_DATA[1],$LOAD=LOAD_DATA[1],$VEL.CP = 2

Halt
             US_PickApproach[1,2] = US_Pick[1,2]
            US_PickApproach[1,2].Z = US_PickApproach[1,2].Z + 100
            US_PickApproachSlow[1,2].Z = US_PickApproach[1,2].Z - 65
            US_Pick1[1,2]= US_Pick[1,2]
            US_Pick2[1,2]= US_Pick[1,2]
            US_Pick3[1,2]= US_Pick[1,2]
            US_Pick1[1,2].X = US_Pick[1,2].X + 0.009187222
            US_Pick1[1,2].Y = US_Pick[1,2].Y  -0.805848
            US_Pick1[1,2].Z = US_Pick[1,2].Z + 0.81393918
            US_Pick1[1,2].A = US_Pick[1,2].A + 0.00272370000000421
            US_Pick1[1,2].B = US_Pick[1,2].B -0.999994156
            US_Pick1[1,2].C = US_Pick[1,2].C -0.00344900000001758
            US_Pick2[1,2].X = US_Pick[1,2].X -1.830273332
            US_Pick2[1,2].Y = US_Pick[1,2].Y  + 0.118088
            US_Pick2[1,2].Z = US_Pick[1,2].Z + 0.22346
            US_Pick2[1,2].A = US_Pick[1,2].A + 0.00272370000000421
            US_Pick2[1,2].B = US_Pick[1,2].B -0.999994156
            US_Pick2[1,2].C = US_Pick[1,2].C -0.00344900000001758
            US_Pick3[1,2].X = US_Pick[1,2].X + 0.764676273
            US_Pick3[1,2].Y = US_Pick[1,2].Y  -1.519576
            US_Pick3[1,2].Z = US_Pick[1,2].Z -0.17324344
            US_Pick3[1,2].A = US_Pick[1,2].A + 0.00272370000000421
            US_Pick3[1,2].B = US_Pick[1,2].B -0.999990132
            US_Pick3[1,2].C = US_Pick[1,2].C -0.00344900000001758
 RtoPLC_BlankCupAVac=False
RtoPLC_BlankCupBVac=False
RtoPLC_BlankCupABlow=False
RtoPLC_BlankCupBBlow=False
 SPTP US_PickApproach[1,2] with $TOOL=TOOL_DATA[1],$BASE=BASE_DATA[1],$LOAD=LOAD_DATA[1],$VEL.CP = 2
 SLIN US_PickApproachSlow[1,2] with $TOOL=TOOL_DATA[1],$BASE=BASE_DATA[1],$LOAD=LOAD_DATA[1],$VEL.CP = 2
 SLIN US_Pick1[1,2] with $TOOL=TOOL_DATA[1],$BASE=BASE_DATA[1],$LOAD=LOAD_DATA[1],$VEL.CP = .01
 SLIN US_Pick2[1,2] with $TOOL=TOOL_DATA[1],$BASE=BASE_DATA[1],$LOAD=LOAD_DATA[1],$VEL.CP = 1
 SLIN US_Pick3[1,2] with $TOOL=TOOL_DATA[1],$BASE=BASE_DATA[1],$LOAD=LOAD_DATA[1],$VEL.CP = 1
 SLIN US_Pick[1,2] with $TOOL=TOOL_DATA[1],$BASE=BASE_DATA[1],$LOAD=LOAD_DATA[1],$VEL.CP = 1

RtoPLC_BlankCupAVac=True
RtoPLC_BlankCupBVac=True
SLIN US_PickApproachSlow[1,2] with $TOOL=TOOL_DATA[1],$BASE=BASE_DATA[1],$LOAD=LOAD_DATA[1],$VEL.CP = 2

Halt

            US_PickApproach[1,3] = US_Pick[1,3]
            US_PickApproach[1,3].Z = US_PickApproach[1,3].Z + 100
            US_PickApproachSlow[1,3].Z = US_PickApproach[1,3].Z - 65
            US_Pick1[1,3]= US_Pick[1,3]
            US_Pick2[1,3]= US_Pick[1,3]
            US_Pick3[1,3]= US_Pick[1,3]
            US_Pick1[1,3].X = US_Pick[1,3].X + 2

            US_Pick1[1,3].Y = US_Pick[1,3].Y  +1


            US_Pick1[1,3].Z = US_Pick[1,3].Z + 0.2
            US_Pick1[1,3].A = US_Pick[1,3].A + 0.00272370000000421
            US_Pick1[1,3].B = US_Pick[1,3].B -0.999994156
            US_Pick1[1,3].C = US_Pick[1,3].C -0.00344900000001758
            US_Pick2[1,3].X = US_Pick[1,3].X -1.830273332
            US_Pick2[1,3].Y = US_Pick[1,3].Y  + 0.118088
            US_Pick2[1,3].Z = US_Pick[1,3].Z + 0.22346
            US_Pick2[1,3].A = US_Pick[1,3].A + 0.00272370000000421
            US_Pick2[1,3].B = US_Pick[1,3].B -0.999994156
            US_Pick2[1,3].C = US_Pick[1,3].C -0.00344900000001758
            US_Pick3[1,3].X = US_Pick[1,3].X + 0.764676273
            US_Pick3[1,3].Y = US_Pick[1,3].Y  -1.519576
            US_Pick3[1,3].Z = US_Pick[1,3].Z -0.17324344
            US_Pick3[1,3].A = US_Pick[1,3].A + 0.00272370000000421
            US_Pick3[1,3].B = US_Pick[1,3].B -0.999990132
            US_Pick3[1,3].C = US_Pick[1,3].C -0.00344900000001758

  RtoPLC_BlankCupAVac=False
RtoPLC_BlankCupBVac=False
RtoPLC_BlankCupABlow=False
RtoPLC_BlankCupBBlow=False
 SPTP US_PickApproach[1,3] with $TOOL=TOOL_DATA[1],$BASE=BASE_DATA[1],$LOAD=LOAD_DATA[1],$VEL.CP = 2
 SLIN US_PickApproachSlow[1,3] with $TOOL=TOOL_DATA[1],$BASE=BASE_DATA[1],$LOAD=LOAD_DATA[1],$VEL.CP = 2
 SLIN US_Pick1[1,3] with $TOOL=TOOL_DATA[1],$BASE=BASE_DATA[1],$LOAD=LOAD_DATA[1],$VEL.CP = .01
 SLIN US_Pick2[1,3] with $TOOL=TOOL_DATA[1],$BASE=BASE_DATA[1],$LOAD=LOAD_DATA[1],$VEL.CP = 1
 SLIN US_Pick3[1,3] with $TOOL=TOOL_DATA[1],$BASE=BASE_DATA[1],$LOAD=LOAD_DATA[1],$VEL.CP = 1
 SLIN US_Pick[1,3] with $TOOL=TOOL_DATA[1],$BASE=BASE_DATA[1],$LOAD=LOAD_DATA[1],$VEL.CP = 1

RtoPLC_BlankCupAVac=True
RtoPLC_BlankCupBVac=True
SLIN US_PickApproachSlow[1,3] with $TOOL=TOOL_DATA[1],$BASE=BASE_DATA[1],$LOAD=LOAD_DATA[1],$VEL.CP = 2

Halt
             US_PickApproach[1,4] = US_Pick[1,4]
            US_PickApproach[1,4].Z = US_PickApproach[1,4].Z + 100
            US_PickApproachSlow[1,4].Z = US_PickApproach[1,4].Z - 65
            US_Pick1[1,4]= US_Pick[1,4]
            US_Pick2[1,4]= US_Pick[1,4]
            US_Pick3[1,4]= US_Pick[1,4]
            US_Pick1[1,4].X = US_Pick[1,4].X + 0.009187222
            US_Pick1[1,4].Y = US_Pick[1,4].Y  -0.805848
            US_Pick1[1,4].Z = US_Pick[1,4].Z + 0.81393918
            US_Pick1[1,4].A = US_Pick[1,4].A + 0.00272370000000421
            US_Pick1[1,4].B = US_Pick[1,4].B -0.999994156
            US_Pick1[1,4].C = US_Pick[1,4].C -0.00344900000001758
            US_Pick2[1,4].X = US_Pick[1,4].X -1.830273332
            US_Pick2[1,4].Y = US_Pick[1,4].Y  + 0.118088
            US_Pick2[1,4].Z = US_Pick[1,4].Z + 0.22346
            US_Pick2[1,4].A = US_Pick[1,4].A + 0.00272370000000421
            US_Pick2[1,4].B = US_Pick[1,4].B -0.999994156
            US_Pick2[1,4].C = US_Pick[1,4].C -0.00344900000001758
            US_Pick3[1,4].X = US_Pick[1,4].X + 0.764676273
            US_Pick3[1,4].Y = US_Pick[1,4].Y  -1.519576
            US_Pick3[1,4].Z = US_Pick[1,4].Z -0.17324344
            US_Pick3[1,4].A = US_Pick[1,4].A + 0.00272370000000421
            US_Pick3[1,4].B = US_Pick[1,4].B -0.999990132
            US_Pick3[1,4].C = US_Pick[1,4].C -0.00344900000001758

  RtoPLC_BlankCupAVac=False
RtoPLC_BlankCupBVac=False
RtoPLC_BlankCupABlow=False
RtoPLC_BlankCupBBlow=False
 SPTP US_PickApproach[1,4] with $TOOL=TOOL_DATA[1],$BASE=BASE_DATA[1],$LOAD=LOAD_DATA[1],$VEL.CP = 2
 SLIN US_PickApproachSlow[1,4] with $TOOL=TOOL_DATA[1],$BASE=BASE_DATA[1],$LOAD=LOAD_DATA[1],$VEL.CP = 2
 SLIN US_Pick1[1,4] with $TOOL=TOOL_DATA[1],$BASE=BASE_DATA[1],$LOAD=LOAD_DATA[1],$VEL.CP = .01
 SLIN US_Pick2[1,4] with $TOOL=TOOL_DATA[1],$BASE=BASE_DATA[1],$LOAD=LOAD_DATA[1],$VEL.CP = 1
 SLIN US_Pick3[1,4] with $TOOL=TOOL_DATA[1],$BASE=BASE_DATA[1],$LOAD=LOAD_DATA[1],$VEL.CP = 1
 SLIN US_Pick[1,4] with $TOOL=TOOL_DATA[1],$BASE=BASE_DATA[1],$LOAD=LOAD_DATA[1],$VEL.CP = 1

RtoPLC_BlankCupAVac=True
RtoPLC_BlankCupBVac=True
SLIN US_PickApproachSlow[1,4] with $TOOL=TOOL_DATA[1],$BASE=BASE_DATA[1],$LOAD=LOAD_DATA[1],$VEL.CP = 2

   US_PickApproach[2,1] = US_Pick[2,1]
            US_PickApproach[2,1].Z = US_PickApproach[2,1].Z + 100
            US_PickApproachSlow[2,1].Z = US_PickApproach[2,1].Z - 65
            US_Pick1[2,1]= US_Pick[2,1]
            US_Pick2[2,1]= US_Pick[2,1]
            US_Pick3[2,1]= US_Pick[2,1]
            US_Pick1[2,1].X = US_Pick[2,1].X + 0.009187222
            US_Pick1[2,1].Y = US_Pick[2,1].Y  -0.805848
            US_Pick1[2,1].Z = US_Pick[2,1].Z + 0.81393918
            US_Pick1[2,1].A = US_Pick[2,1].A + 0.00272370000000421
            US_Pick1[2,1].B = US_Pick[2,1].B -0.999994156
            US_Pick1[2,1].C = US_Pick[2,1].C -0.00344900000001758
            US_Pick2[2,1].X = US_Pick[2,1].X -1.830273332
            US_Pick2[2,1].Y = US_Pick[2,1].Y  + 0.118088
            US_Pick2[2,1].Z = US_Pick[2,1].Z + 0.22346
            US_Pick2[2,1].A = US_Pick[2,1].A + 0.00272370000000421
            US_Pick2[2,1].B = US_Pick[2,1].B -0.999994156
            US_Pick2[2,1].C = US_Pick[2,1].C -0.00344900000001758
            US_Pick3[2,1].X = US_Pick[2,1].X + 0.764676273
            US_Pick3[2,1].Y = US_Pick[2,1].Y  -1.519576
            US_Pick3[2,1].Z = US_Pick[2,1].Z -0.17324344
            US_Pick3[2,1].A = US_Pick[2,1].A + 0.00272370000000421
            US_Pick3[2,1].B = US_Pick[2,1].B -0.999990132
            US_Pick3[2,1].C = US_Pick[2,1].C -0.00344900000001758
 RtoPLC_BlankCupAVac=False
RtoPLC_BlankCupBVac=False
RtoPLC_BlankCupABlow=False
RtoPLC_BlankCupBBlow=False
 SPTP US_PickApproach[2,1] with $TOOL=TOOL_DATA[1],$BASE=BASE_DATA[1],$LOAD=LOAD_DATA[1],$VEL.CP = 2
 SLIN US_PickApproachSlow[2,1] with $TOOL=TOOL_DATA[1],$BASE=BASE_DATA[1],$LOAD=LOAD_DATA[1],$VEL.CP = 2
 SLIN US_Pick1[2,1] with $TOOL=TOOL_DATA[1],$BASE=BASE_DATA[1],$LOAD=LOAD_DATA[1],$VEL.CP = .01
 SLIN US_Pick2[2,1] with $TOOL=TOOL_DATA[1],$BASE=BASE_DATA[1],$LOAD=LOAD_DATA[1],$VEL.CP = 1
 SLIN US_Pick3[2,1] with $TOOL=TOOL_DATA[1],$BASE=BASE_DATA[1],$LOAD=LOAD_DATA[1],$VEL.CP = 1
 SLIN US_Pick[2,1] with $TOOL=TOOL_DATA[1],$BASE=BASE_DATA[1],$LOAD=LOAD_DATA[1],$VEL.CP = 1

RtoPLC_BlankCupAVac=True
RtoPLC_BlankCupBVac=True
SLIN US_PickApproachSlow[2,1] with $TOOL=TOOL_DATA[1],$BASE=BASE_DATA[1],$LOAD=LOAD_DATA[1],$VEL.CP = 2

Halt
             US_PickApproach[2,2] = US_Pick[2,2]
            US_PickApproach[2,2].Z = US_PickApproach[2,2].Z + 100
            US_PickApproachSlow[2,2].Z = US_PickApproach[2,2].Z - 65
            US_Pick1[2,2]= US_Pick[2,2]
            US_Pick2[2,2]= US_Pick[2,2]
            US_Pick3[2,2]= US_Pick[2,2]
            US_Pick1[2,2].X = US_Pick[2,2].X + 0.009187222
            US_Pick1[2,2].Y = US_Pick[2,2].Y  -0.805848
            US_Pick1[2,2].Z = US_Pick[2,2].Z + 0.81393918
            US_Pick1[2,2].A = US_Pick[2,2].A + 0.00272370000000421
            US_Pick1[2,2].B = US_Pick[2,2].B -0.999994156
            US_Pick1[2,2].C = US_Pick[2,2].C -0.00344900000001758
            US_Pick2[2,2].X = US_Pick[2,2].X -1.830273332
            US_Pick2[2,2].Y = US_Pick[2,2].Y  + 0.118088
            US_Pick2[2,2].Z = US_Pick[2,2].Z + 0.22346
            US_Pick2[2,2].A = US_Pick[2,2].A + 0.00272370000000421
            US_Pick2[2,2].B = US_Pick[2,2].B -0.999994156
            US_Pick2[2,2].C = US_Pick[2,2].C -0.00344900000001758
            US_Pick3[2,2].X = US_Pick[2,2].X + 0.764676273
            US_Pick3[2,2].Y = US_Pick[2,2].Y  -1.519576
            US_Pick3[2,2].Z = US_Pick[2,2].Z -0.17324344
            US_Pick3[2,2].A = US_Pick[2,2].A + 0.00272370000000421
            US_Pick3[2,2].B = US_Pick[2,2].B -0.999990132
            US_Pick3[2,2].C = US_Pick[2,2].C -0.00344900000001758
 RtoPLC_BlankCupAVac=False
RtoPLC_BlankCupBVac=False
RtoPLC_BlankCupABlow=False
RtoPLC_BlankCupBBlow=False
 SPTP US_PickApproach[2,2] with $TOOL=TOOL_DATA[1],$BASE=BASE_DATA[1],$LOAD=LOAD_DATA[1],$VEL.CP = 2
 SLIN US_PickApproachSlow[2,2] with $TOOL=TOOL_DATA[1],$BASE=BASE_DATA[1],$LOAD=LOAD_DATA[1],$VEL.CP = 2
 SLIN US_Pick1[2,2] with $TOOL=TOOL_DATA[1],$BASE=BASE_DATA[1],$LOAD=LOAD_DATA[1],$VEL.CP = .01
 SLIN US_Pick2[2,2] with $TOOL=TOOL_DATA[1],$BASE=BASE_DATA[1],$LOAD=LOAD_DATA[1],$VEL.CP = 1
 SLIN US_Pick3[2,2] with $TOOL=TOOL_DATA[1],$BASE=BASE_DATA[1],$LOAD=LOAD_DATA[1],$VEL.CP = 1
 SLIN US_Pick[2,2] with $TOOL=TOOL_DATA[1],$BASE=BASE_DATA[1],$LOAD=LOAD_DATA[1],$VEL.CP = 1

RtoPLC_BlankCupAVac=True
RtoPLC_BlankCupBVac=True
SLIN US_PickApproachSlow[2,2] with $TOOL=TOOL_DATA[1],$BASE=BASE_DATA[1],$LOAD=LOAD_DATA[1],$VEL.CP = 2

Halt
            US_PickApproach[2,3] = US_Pick[2,3]
            US_PickApproach[2,3].Z = US_PickApproach[2,3].Z + 100
            US_PickApproachSlow[2,3].Z = US_PickApproach[2,3].Z - 65
            US_Pick1[2,3]= US_Pick[2,3]
            US_Pick2[2,3]= US_Pick[2,3]
            US_Pick3[2,3]= US_Pick[2,3]
            US_Pick1[2,3].X = US_Pick[2,3].X + 0.009187222
            US_Pick1[2,3].Y = US_Pick[2,3].Y  -0.805848
            US_Pick1[2,3].Z = US_Pick[2,3].Z + 0.81393918
            US_Pick1[2,3].A = US_Pick[2,3].A + 0.00272370000000421
            US_Pick1[2,3].B = US_Pick[2,3].B -0.999994156
            US_Pick1[2,3].C = US_Pick[2,3].C -0.00344900000001758
            US_Pick2[2,3].X = US_Pick[2,3].X -1.830273332
            US_Pick2[2,3].Y = US_Pick[2,3].Y  + 0.118088
            US_Pick2[2,3].Z = US_Pick[2,3].Z + 0.22346
            US_Pick2[2,3].A = US_Pick[2,3].A + 0.00272370000000421
            US_Pick2[2,3].B = US_Pick[2,3].B -0.999994156
            US_Pick2[2,3].C = US_Pick[2,3].C -0.00344900000001758
            US_Pick3[2,3].X = US_Pick[2,3].X + 0.764676273
            US_Pick3[2,3].Y = US_Pick[2,3].Y  -1.519576
            US_Pick3[2,3].Z = US_Pick[2,3].Z -0.17324344
            US_Pick3[2,3].A = US_Pick[2,3].A + 0.00272370000000421
            US_Pick3[2,3].B = US_Pick[2,3].B -0.999990132
            US_Pick3[2,3].C = US_Pick[2,3].C -0.00344900000001758

  RtoPLC_BlankCupAVac=False
RtoPLC_BlankCupBVac=False
RtoPLC_BlankCupABlow=False
RtoPLC_BlankCupBBlow=False
 SPTP US_PickApproach[2,3] with $TOOL=TOOL_DATA[1],$BASE=BASE_DATA[1],$LOAD=LOAD_DATA[1],$VEL.CP = 2
 SLIN US_PickApproachSlow[2,3] with $TOOL=TOOL_DATA[1],$BASE=BASE_DATA[1],$LOAD=LOAD_DATA[1],$VEL.CP = 2
 SLIN US_Pick1[2,3] with $TOOL=TOOL_DATA[1],$BASE=BASE_DATA[1],$LOAD=LOAD_DATA[1],$VEL.CP = .01
 SLIN US_Pick2[2,3] with $TOOL=TOOL_DATA[1],$BASE=BASE_DATA[1],$LOAD=LOAD_DATA[1],$VEL.CP = 1
 SLIN US_Pick3[2,3] with $TOOL=TOOL_DATA[1],$BASE=BASE_DATA[1],$LOAD=LOAD_DATA[1],$VEL.CP = 1
 SLIN US_Pick[2,3] with $TOOL=TOOL_DATA[1],$BASE=BASE_DATA[1],$LOAD=LOAD_DATA[1],$VEL.CP = 1

RtoPLC_BlankCupAVac=True
RtoPLC_BlankCupBVac=True
SLIN US_PickApproachSlow[2,3] with $TOOL=TOOL_DATA[1],$BASE=BASE_DATA[1],$LOAD=LOAD_DATA[1],$VEL.CP = 2

Halt
             US_PickApproach[2,4] = US_Pick[2,4]
            US_PickApproach[2,4].Z = US_PickApproach[2,4].Z + 100
            US_PickApproachSlow[2,4].Z = US_PickApproach[2,4].Z - 65
            US_Pick1[2,4]= US_Pick[2,4]
            US_Pick2[2,4]= US_Pick[2,4]
            US_Pick3[2,4]= US_Pick[2,4]
            US_Pick1[2,4].X = US_Pick[2,4].X + 0.009187222
            US_Pick1[2,4].Y = US_Pick[2,4].Y  -0.805848
            US_Pick1[2,4].Z = US_Pick[2,4].Z + 0.81393918
            US_Pick1[2,4].A = US_Pick[2,4].A + 0.00272370000000421
            US_Pick1[2,4].B = US_Pick[2,4].B -0.999994156
            US_Pick1[2,4].C = US_Pick[2,4].C -0.00344900000001758
            US_Pick2[2,4].X = US_Pick[2,4].X -1.830273332
            US_Pick2[2,4].Y = US_Pick[2,4].Y  + 0.118088
            US_Pick2[2,4].Z = US_Pick[2,4].Z + 0.22346
            US_Pick2[2,4].A = US_Pick[2,4].A + 0.00272370000000421
            US_Pick2[2,4].B = US_Pick[2,4].B -0.999994156
            US_Pick2[2,4].C = US_Pick[2,4].C -0.00344900000001758
            US_Pick3[2,4].X = US_Pick[2,4].X + 0.764676273
            US_Pick3[2,4].Y = US_Pick[2,4].Y  -1.519576
            US_Pick3[2,4].Z = US_Pick[2,4].Z -0.17324344
            US_Pick3[2,4].A = US_Pick[2,4].A + 0.00272370000000421
            US_Pick3[2,4].B = US_Pick[2,4].B -0.999990132
            US_Pick3[2,4].C = US_Pick[2,4].C -0.00344900000001758

  RtoPLC_BlankCupAVac=False
RtoPLC_BlankCupBVac=False
RtoPLC_BlankCupABlow=False
RtoPLC_BlankCupBBlow=False
 SPTP US_PickApproach[2,4] with $TOOL=TOOL_DATA[1],$BASE=BASE_DATA[1],$LOAD=LOAD_DATA[1],$VEL.CP = 2
 SLIN US_PickApproachSlow[2,4] with $TOOL=TOOL_DATA[1],$BASE=BASE_DATA[1],$LOAD=LOAD_DATA[1],$VEL.CP = 2
 SLIN US_Pick1[2,4] with $TOOL=TOOL_DATA[1],$BASE=BASE_DATA[1],$LOAD=LOAD_DATA[1],$VEL.CP = .01
 SLIN US_Pick2[2,4] with $TOOL=TOOL_DATA[1],$BASE=BASE_DATA[1],$LOAD=LOAD_DATA[1],$VEL.CP = 1
 SLIN US_Pick3[2,4] with $TOOL=TOOL_DATA[1],$BASE=BASE_DATA[1],$LOAD=LOAD_DATA[1],$VEL.CP = 1
 SLIN US_Pick[2,4] with $TOOL=TOOL_DATA[1],$BASE=BASE_DATA[1],$LOAD=LOAD_DATA[1],$VEL.CP = 1

RtoPLC_BlankCupAVac=True
RtoPLC_BlankCupBVac=True
SLIN US_PickApproachSlow[2,4] with $TOOL=TOOL_DATA[1],$BASE=BASE_DATA[1],$LOAD=LOAD_DATA[1],$VEL.CP = 2

EndOfModule:
END

--- PickPlaceTrayTeach.dat ---
&ACCESS  RVP
&PARAM DISKPATH = KRC:\R1\Program
&REL 58
DEFDAT  PICKPLACETRAYTEACH
;FOLD EXTERNAL DECLARATIONS;%{PE}%MKUKATPBASIS,%CEXT,%VCOMMON,%P
;FOLD BASISTECH EXT;%{PE}%MKUKATPBASIS,%CEXT,%VEXT,%P
EXT  BAS (BAS_COMMAND  :IN,REAL  :IN )
DECL INT SUCCESS
;ENDFOLD (BASISTECH EXT)
;FOLD USER EXT;%{E}%MKUKATPUSER,%CEXT,%VEXT,%P
;Make your modifications here

;ENDFOLD (USER EXT)
;ENDFOLD (EXTERNAL DECLARATIONS)


DECL LDAT LCPDAT1={VEL 2.00000,ACC 60.0000,APO_DIST 500.000,APO_FAC 50.0000,AXIS_VEL 100.000,AXIS_ACC 60.0000,ORI_TYP #VAR,CIRC_TYP #BASE,JERK_FAC 50.0000,GEAR_JERK 100.000,EXAX_IGN 0}
DECL PDAT PDEFAULT={VEL 100.000,ACC 60.0000,APO_DIST 500.000,APO_MODE #CDIS,GEAR_JERK 100.000,EXAX_IGN 0}
DECL LDAT LCPDAT2={VEL 2.00000,ACC 60.0000,APO_DIST 500.000,APO_FAC 50.0000,AXIS_VEL 100.000,AXIS_ACC 60.0000,ORI_TYP #VAR,CIRC_TYP #BASE,JERK_FAC 50.0000,GEAR_JERK 100.000,EXAX_IGN 0}
DECL PDAT PPDAT1={VEL 100.000,ACC 60.0000,APO_DIST 500.000,APO_MODE #CDIS,GEAR_JERK 100.000,EXAX_IGN 0}
DECL LDAT LCPDAT3={VEL 2.00000,ACC 60.0000,APO_DIST 500.000,APO_FAC 50.0000,AXIS_VEL 100.000,AXIS_ACC 60.0000,ORI_TYP #VAR,CIRC_TYP #BASE,JERK_FAC 50.0000,GEAR_JERK 100.000,EXAX_IGN 0}
DECL LDAT LCPDAT4={VEL 2.00000,ACC 60.0000,APO_DIST 500.000,APO_FAC 50.0000,AXIS_VEL 100.000,AXIS_ACC 60.0000,ORI_TYP #VAR,CIRC_TYP #BASE,JERK_FAC 50.0000,GEAR_JERK 100.000,EXAX_IGN 0}
DECL LDAT LCPDAT5={VEL 2.00000,ACC 60.0000,APO_DIST 500.000,APO_FAC 50.0000,AXIS_VEL 100.000,AXIS_ACC 60.0000,ORI_TYP #VAR,CIRC_TYP #BASE,JERK_FAC 50.0000,GEAR_JERK 100.000,EXAX_IGN 0}
DECL PDAT PPDAT2={VEL 100.000,ACC 60.0000,APO_DIST 500.000,APO_MODE #CDIS,GEAR_JERK 100.000,EXAX_IGN 0}
DECL PDAT PPDAT3={VEL 100.000,ACC 60.0000,APO_DIST 500.000,APO_MODE #CDIS,GEAR_JERK 100.000,EXAX_IGN 0}
DECL PDAT PPDAT4={VEL 100.000,ACC 60.0000,APO_DIST 500.000,APO_MODE #CDIS,GEAR_JERK 100.000,EXAX_IGN 0}
DECL E6POS XUS_A1Turn={X -108.546844,Y -232.779465,Z 1087.90991,A 64.9999619,B 35.0000,C 179.999985,S 2,T 34,E1 0.0,E2 0.0,E3 0.0,E4 0.0,E5 0.0,E6 0.0}
DECL FDAT FUS_A1Turn={TOOL_NO 0,BASE_NO 0,IPO_FRAME #BASE,POINT2[] " "}
DECL E6POS XUS_A1Return={X -108.546844,Y -232.779465,Z 1087.90991,A 64.9999619,B 35.0000,C 179.999985,S 2,T 34,E1 0.0,E2 0.0,E3 0.0,E4 0.0,E5 0.0,E6 0.0}
DECL FDAT FUS_A1Return={TOOL_NO 0,BASE_NO 0,IPO_FRAME #BASE,POINT2[] " "}
DECL LDAT LCPDAT6={VEL 2.00000,ACC 60.0000,APO_DIST 500.000,APO_FAC 50.0000,AXIS_VEL 100.000,AXIS_ACC 60.0000,ORI_TYP #VAR,CIRC_TYP #BASE,JERK_FAC 50.0000,GEAR_JERK 100.000,EXAX_IGN 0}
DECL LDAT LCPDAT7={VEL 2.00000,ACC 60.0000,APO_DIST 500.000,APO_FAC 50.0000,AXIS_VEL 100.000,AXIS_ACC 60.0000,ORI_TYP #VAR,CIRC_TYP #BASE,JERK_FAC 50.0000,GEAR_JERK 100.000,EXAX_IGN 0}
DECL LDAT LCPDAT8={VEL 0.200000,ACC 60.0000,APO_DIST 500.000,APO_FAC 50.0000,AXIS_VEL 100.000,AXIS_ACC 60.0000,ORI_TYP #VAR,CIRC_TYP #BASE,JERK_FAC 50.0000,GEAR_JERK 100.000,EXAX_IGN 0}
DECL LDAT LCPDAT9={VEL 0.200000,ACC 60.0000,APO_DIST 500.000,APO_FAC 50.0000,AXIS_VEL 100.000,AXIS_ACC 60.0000,ORI_TYP #VAR,CIRC_TYP #BASE,JERK_FAC 50.0000,GEAR_JERK 100.000,EXAX_IGN 0}
DECL LDAT LCPDAT10={VEL 0.200000,ACC 60.0000,APO_DIST 500.000,APO_FAC 50.0000,AXIS_VEL 100.000,AXIS_ACC 60.0000,ORI_TYP #VAR,CIRC_TYP #BASE,JERK_FAC 50.0000,GEAR_JERK 100.000,EXAX_IGN 0}
DECL E6POS XUS_TraySlideAppr={X 362.802795,Y 241.343796,Z 97.5473,A -0.00488100,B 0.488478,C -0.0135530,S 2,T 2,E1 0.0,E2 0.0,E3 0.0,E4 0.0,E5 0.0,E6 0.0}
DECL FDAT FUS_TraySlideAppr={TOOL_NO 3,BASE_NO 6,IPO_FRAME #BASE,POINT2[] " "}
DECL E6POS XUS_TraySlide={X 361.950256,Y 241.320206,Z -2.44906306,A -0.00488100,B 0.488478,C -0.0135530,S 2,T 2,E1 0.0,E2 0.0,E3 0.0,E4 0.0,E5 0.0,E6 0.0}
DECL FDAT FUS_TraySlide={TOOL_NO 3,BASE_NO 6,IPO_FRAME #BASE,POINT2[] " "}
DECL E6POS XUS_TraySlideReturn={X 985.080200,Y 241.290787,Z 92.2419128,A -0.00488100,B 0.488478,C -0.0135530,S 2,T 2,E1 0.0,E2 0.0,E3 0.0,E4 0.0,E5 0.0,E6 0.0}
DECL FDAT FUS_TraySlideReturn={TOOL_NO 3,BASE_NO 6,IPO_FRAME #BASE,POINT2[] " "}
DECL E6POS XUS_TraySlideEnd={X 984.227661,Y 241.267303,Z -7.75470400,A -0.00487200,B 0.488485,C -0.0135230,S 2,T 2,E1 0.0,E2 0.0,E3 0.0,E4 0.0,E5 0.0,E6 0.0}
DECL FDAT FUS_TraySlideEnd={TOOL_NO 3,BASE_NO 6,IPO_FRAME #BASE,POINT2[] " "}
DECL PDAT PPDAT5={VEL 100.000,ACC 60.0000,APO_DIST 500.000,APO_MODE #CDIS,GEAR_JERK 100.000,EXAX_IGN 0}
DECL E6POS XDS_A1Turn={X 44.6004448,Y -252.941681,Z 1087.90991,A 99.9999619,B 35.0000,C 179.999985,S 2,T 34,E1 0.0,E2 0.0,E3 0.0,E4 0.0,E5 0.0,E6 0.0}
DECL FDAT FDS_A1Turn={TOOL_NO 0,BASE_NO 0,IPO_FRAME #BASE,POINT2[] " "}

DECL PDAT PPDAT11={VEL 100.000,ACC 60.0000,APO_DIST 500.000,APO_MODE #CDIS,GEAR_JERK 100.000,EXAX_IGN 0}



DECL PDAT PPDAT6={VEL 100.000,ACC 60.0000,APO_DIST 500.000,APO_MODE #CDIS,GEAR_JERK 100.000,EXAX_IGN 0}
DECL MODULEPARAM_T LAST_TP_PARAMS={PARAMS[] "Kuka.VelocityFieldEnabled=True; Kuka.ColDetectFieldEnabled=True; Kuka.MovementParameterFieldEnabled=True; Kuka.IsAngleEnabled=False; Kuka.PointName=DS_TeachPick2_4; Kuka.FrameData.base_no=5; Kuka.FrameData.tool_no=2; Kuka.FrameData.ipo_frame=#BASE; Kuka.isglobalpoint=False; Kuka.MoveDataPtpName=PDAT12; Kuka.MovementDataPdat.apo_mode=#CDIS; Kuka.MovementDataPdat.apo_dist=500; Kuka.MovementData.vel=1; Kuka.MovementData.acc=100; Kuka.MovementData.exax_ign=0; Kuka.VelocityPtp=100; Kuka.BlendingEnabled=False; Kuka.APXEnabled=False; Kuka.CurrentCDSetIndex=0; Kuka.FrameData.point2=; Kuka.MoveDataName=CPDAT25; Kuka.MovementData.cb={AUX_PT {ORI #CONSIDER,E1 #CONSIDER,E2 #CONSIDER,E3 #CONSIDER,E4 #CONSIDER,E5 #CONSIDER,E6 #CONSIDER},TARGET_PT {ORI #INTERPOLATE,E1 #INTERPOLATE,E2 #INTERPOLATE,E3 #INTERPOLATE,E4 #INTERPOLATE,E5 #INTERPOLATE,E6 #INTERPOLATE}}; Kuka.MovementData.apo_fac=50; Kuka.MovementData.apo_dist=500; Kuka.MovementData.axis_acc=100; Kuka.MovementData.axis_vel=100; Kuka.MovementData.circ_typ=#BASE; Kuka.MovementData.jerk_fac=50; Kuka.MovementData.ori_typ=#VAR; Kuka.VelocityPath=1    "}
DECL PDAT PPDAT7={VEL 100.000,ACC 60.0000,APO_DIST 500.000,APO_MODE #CDIS,GEAR_JERK 100.000,EXAX_IGN 0}
DECL FDAT FUS_TeachPick={TOOL_NO 1,BASE_NO 1,IPO_FRAME #BASE,POINT2[] " "}
DECL E6POS XUS_TeachPick={X 0.871399701,Y 179.209305,Z 5.35049486,A 90.9870224,B 0.454473257,C -179.703384,S 2,T 34,E1 0.0,E2 0.0,E3 0.0,E4 0.0,E5 0.0,E6 0.0}
DECL LDAT LCPDAT01={VEL 2.00000,ACC 60.0000,APO_DIST 500.000,APO_FAC 50.0000,AXIS_VEL 100.000,AXIS_ACC 60.0000,ORI_TYP #VAR,CIRC_TYP #BASE,JERK_FAC 50.0000,GEAR_JERK 100.000,EXAX_IGN 0,CB {AUX_PT {ORI #CONSIDER,E1 #CONSIDER,E2 #CONSIDER,E3 #CONSIDER,E4 #CONSIDER,E5 #CONSIDER,E6 #CONSIDER},TARGET_PT {ORI #INTERPOLATE,E1 #INTERPOLATE,E2 #INTERPOLATE,E3 #INTERPOLATE,E4 #INTERPOLATE,E5 #INTERPOLATE,E6 #INTERPOLATE}}}
DECL E6POS US_PickApproach_1[2,4]
DECL E6POS US_PickApproachSlow_1[1,1]
DECL LDAT LCPDAT02={VEL 0.200000,ACC 60.0000,APO_DIST 500.000,APO_FAC 50.0000,AXIS_VEL 100.000,AXIS_ACC 60.0000,ORI_TYP #VAR,CIRC_TYP #BASE,JERK_FAC 50.0000,GEAR_JERK 100.000,EXAX_IGN 0,CB {AUX_PT {ORI #CONSIDER,E1 #CONSIDER,E2 #CONSIDER,E3 #CONSIDER,E4 #CONSIDER,E5 #CONSIDER,E6 #CONSIDER},TARGET_PT {ORI #INTERPOLATE,E1 #INTERPOLATE,E2 #INTERPOLATE,E3 #INTERPOLATE,E4 #INTERPOLATE,E5 #INTERPOLATE,E6 #INTERPOLATE}}}
DECL LDAT LCPDAT03={VEL 0.200000,ACC 60.0000,APO_DIST 500.000,APO_FAC 50.0000,AXIS_VEL 100.000,AXIS_ACC 60.0000,ORI_TYP #VAR,CIRC_TYP #BASE,JERK_FAC 50.0000,GEAR_JERK 100.000,EXAX_IGN 0,CB {AUX_PT {ORI #CONSIDER,E1 #CONSIDER,E2 #CONSIDER,E3 #CONSIDER,E4 #CONSIDER,E5 #CONSIDER,E6 #CONSIDER},TARGET_PT {ORI #INTERPOLATE,E1 #INTERPOLATE,E2 #INTERPOLATE,E3 #INTERPOLATE,E4 #INTERPOLATE,E5 #INTERPOLATE,E6 #INTERPOLATE}}}
DECL E6POS XUS_TeachPick1={X 0.927678406,Y 183.215424,Z 5.87333918,A 90.0619583,B 0.366831064,C 179.842010,S 2,T 34,E1 0.0,E2 0.0,E3 0.0,E4 0.0,E5 0.0,E6 0.0}
DECL FDAT FUS_TeachPick1={TOOL_NO 1,BASE_NO 1,IPO_FRAME #BASE,POINT2[] " "}
DECL LDAT LCPDAT04={VEL 1.00000,ACC 60.0000,APO_DIST 500.000,APO_FAC 50.0000,AXIS_VEL 100.000,AXIS_ACC 60.0000,ORI_TYP #VAR,CIRC_TYP #BASE,JERK_FAC 50.0000,GEAR_JERK 100.000,EXAX_IGN 0,CB {AUX_PT {ORI #CONSIDER,E1 #CONSIDER,E2 #CONSIDER,E3 #CONSIDER,E4 #CONSIDER,E5 #CONSIDER,E6 #CONSIDER},TARGET_PT {ORI #INTERPOLATE,E1 #INTERPOLATE,E2 #INTERPOLATE,E3 #INTERPOLATE,E4 #INTERPOLATE,E5 #INTERPOLATE,E6 #INTERPOLATE}}}
DECL E6POS XUS_TeachPick2={X 2.76713896,Y 182.527664,Z 5.28286,A 90.0619583,B 0.366831064,C 179.842010,S 2,T 34,E1 0.0,E2 0.0,E3 0.0,E4 0.0,E5 0.0,E6 0.0}
DECL FDAT FUS_TeachPick2={TOOL_NO 1,BASE_NO 1,IPO_FRAME #BASE,POINT2[] " "}
DECL LDAT LCPDAT05={VEL 1.00000,ACC 60.0000,APO_DIST 500.000,APO_FAC 50.0000,AXIS_VEL 100.000,AXIS_ACC 60.0000,ORI_TYP #VAR,CIRC_TYP #BASE,JERK_FAC 50.0000,GEAR_JERK 100.000,EXAX_IGN 0,CB {AUX_PT {ORI #CONSIDER,E1 #CONSIDER,E2 #CONSIDER,E3 #CONSIDER,E4 #CONSIDER,E5 #CONSIDER,E6 #CONSIDER},TARGET_PT {ORI #INTERPOLATE,E1 #INTERPOLATE,E2 #INTERPOLATE,E3 #INTERPOLATE,E4 #INTERPOLATE,E5 #INTERPOLATE,E6 #INTERPOLATE}}}
DECL E6POS XUS_TeachPick3={X 0.172189355,Y 180.890,Z 4.88615656,A 90.0619583,B 0.366835088,C 179.842010,S 2,T 34,E1 0.0,E2 0.0,E3 0.0,E4 0.0,E5 0.0,E6 0.0}
DECL FDAT FUS_TeachPick3={TOOL_NO 1,BASE_NO 1,IPO_FRAME #BASE,POINT2[] " "}
DECL LDAT LCPDAT06={VEL 1.00000,ACC 60.0000,APO_DIST 500.000,APO_FAC 50.0000,AXIS_VEL 100.000,AXIS_ACC 60.0000,ORI_TYP #VAR,CIRC_TYP #BASE,JERK_FAC 50.0000,GEAR_JERK 100.000,EXAX_IGN 0,CB {AUX_PT {ORI #CONSIDER,E1 #CONSIDER,E2 #CONSIDER,E3 #CONSIDER,E4 #CONSIDER,E5 #CONSIDER,E6 #CONSIDER},TARGET_PT {ORI #INTERPOLATE,E1 #INTERPOLATE,E2 #INTERPOLATE,E3 #INTERPOLATE,E4 #INTERPOLATE,E5 #INTERPOLATE,E6 #INTERPOLATE}}}
DECL E6POS XUS_TeachPick1_2={X 51.9155083,Y 180.086395,Z 5.05748510,A 90.9870224,B 0.454473138,C -179.703384,S 2,T 34,E1 0.0,E2 0.0,E3 0.0,E4 0.0,E5 0.0,E6 0.0}
DECL FDAT FUS_TeachPick1_2={TOOL_NO 1,BASE_NO 1,IPO_FRAME #BASE,POINT2[] " "}
DECL LDAT LCPDAT07={VEL 1.00000,ACC 60.0000,APO_DIST 500.000,APO_FAC 50.0000,AXIS_VEL 100.000,AXIS_ACC 60.0000,ORI_TYP #VAR,CIRC_TYP #BASE,JERK_FAC 50.0000,GEAR_JERK 100.000,EXAX_IGN 0,CB {AUX_PT {ORI #CONSIDER,E1 #CONSIDER,E2 #CONSIDER,E3 #CONSIDER,E4 #CONSIDER,E5 #CONSIDER,E6 #CONSIDER},TARGET_PT {ORI #INTERPOLATE,E1 #INTERPOLATE,E2 #INTERPOLATE,E3 #INTERPOLATE,E4 #INTERPOLATE,E5 #INTERPOLATE,E6 #INTERPOLATE}}}
DECL E6POS XUS_TeachPick1_3={X 204.520859,Y 181.062241,Z 5.48895264,A 91.0696335,B 0.563846171,C -179.516556,S 2,T 34,E1 0.0,E2 0.0,E3 0.0,E4 0.0,E5 0.0,E6 0.0}
DECL FDAT FUS_TeachPick1_3={TOOL_NO 1,BASE_NO 1,IPO_FRAME #BASE,POINT2[] " "}
DECL LDAT LCPDAT08={VEL 1.00000,ACC 60.0000,APO_DIST 500.000,APO_FAC 50.0000,AXIS_VEL 100.000,AXIS_ACC 60.0000,ORI_TYP #VAR,CIRC_TYP #BASE,JERK_FAC 50.0000,GEAR_JERK 100.000,EXAX_IGN 0,CB {AUX_PT {ORI #CONSIDER,E1 #CONSIDER,E2 #CONSIDER,E3 #CONSIDER,E4 #CONSIDER,E5 #CONSIDER,E6 #CONSIDER},TARGET_PT {ORI #INTERPOLATE,E1 #INTERPOLATE,E2 #INTERPOLATE,E3 #INTERPOLATE,E4 #INTERPOLATE,E5 #INTERPOLATE,E6 #INTERPOLATE}}}
DECL E6POS XUS_TeachPick1_4={X 254.713776,Y 181.417389,Z 6.04867649,A 90.8385544,B 0.550665140,C -179.404114,S 2,T 34,E1 0.0,E2 0.0,E3 0.0,E4 0.0,E5 0.0,E6 0.0}
DECL FDAT FUS_TeachPick1_4={TOOL_NO 1,BASE_NO 1,IPO_FRAME #BASE,POINT2[] " "}
DECL LDAT LCPDAT09={VEL 1.00000,ACC 60.0000,APO_DIST 500.000,APO_FAC 50.0000,AXIS_VEL 100.000,AXIS_ACC 60.0000,ORI_TYP #VAR,CIRC_TYP #BASE,JERK_FAC 50.0000,GEAR_JERK 100.000,EXAX_IGN 0,CB {AUX_PT {ORI #CONSIDER,E1 #CONSIDER,E2 #CONSIDER,E3 #CONSIDER,E4 #CONSIDER,E5 #CONSIDER,E6 #CONSIDER},TARGET_PT {ORI #INTERPOLATE,E1 #INTERPOLATE,E2 #INTERPOLATE,E3 #INTERPOLATE,E4 #INTERPOLATE,E5 #INTERPOLATE,E6 #INTERPOLATE}}}
DECL E6POS XUS_TeachPick2_1={X 2.06639624,Y -4.28187561,Z 6.34910250,A 90.6391068,B 0.985694468,C -179.495758,S 2,T 34,E1 0.0,E2 0.0,E3 0.0,E4 0.0,E5 0.0,E6 0.0}
DECL FDAT FUS_TeachPick2_1={TOOL_NO 1,BASE_NO 1,IPO_FRAME #BASE,POINT2[] " "}
DECL LDAT LCPDAT11={VEL 1.00000,ACC 60.0000,APO_DIST 500.000,APO_FAC 50.0000,AXIS_VEL 100.000,AXIS_ACC 60.0000,ORI_TYP #VAR,CIRC_TYP #BASE,JERK_FAC 50.0000,GEAR_JERK 100.000,EXAX_IGN 0,CB {AUX_PT {ORI #CONSIDER,E1 #CONSIDER,E2 #CONSIDER,E3 #CONSIDER,E4 #CONSIDER,E5 #CONSIDER,E6 #CONSIDER},TARGET_PT {ORI #INTERPOLATE,E1 #INTERPOLATE,E2 #INTERPOLATE,E3 #INTERPOLATE,E4 #INTERPOLATE,E5 #INTERPOLATE,E6 #INTERPOLATE}}}
DECL E6POS XUS_TeachPick2_2={X 52.7561111,Y -4.29654837,Z 6.11669302,A 90.6391068,B 0.985694587,C -179.495758,S 2,T 34,E1 0.0,E2 0.0,E3 0.0,E4 0.0,E5 0.0,E6 0.0}
DECL FDAT FUS_TeachPick2_2={TOOL_NO 1,BASE_NO 1,IPO_FRAME #BASE,POINT2[] " "}
DECL LDAT LCPDAT12={VEL 1.00000,ACC 60.0000,APO_DIST 500.000,APO_FAC 50.0000,AXIS_VEL 100.000,AXIS_ACC 60.0000,ORI_TYP #VAR,CIRC_TYP #BASE,JERK_FAC 50.0000,GEAR_JERK 100.000,EXAX_IGN 0,CB {AUX_PT {ORI #CONSIDER,E1 #CONSIDER,E2 #CONSIDER,E3 #CONSIDER,E4 #CONSIDER,E5 #CONSIDER,E6 #CONSIDER},TARGET_PT {ORI #INTERPOLATE,E1 #INTERPOLATE,E2 #INTERPOLATE,E3 #INTERPOLATE,E4 #INTERPOLATE,E5 #INTERPOLATE,E6 #INTERPOLATE}}}
DECL E6POS XUS_TeachPick2_3={X 205.393784,Y -3.18428564,Z 6.22483253,A 90.8425293,B 0.983898520,C -179.492264,S 2,T 34,E1 0.0,E2 0.0,E3 0.0,E4 0.0,E5 0.0,E6 0.0}
DECL FDAT FUS_TeachPick2_3={TOOL_NO 1,BASE_NO 1,IPO_FRAME #BASE,POINT2[] " "}
DECL LDAT LCPDAT13={VEL 1.00000,ACC 60.0000,APO_DIST 500.000,APO_FAC 50.0000,AXIS_VEL 100.000,AXIS_ACC 60.0000,ORI_TYP #VAR,CIRC_TYP #BASE,JERK_FAC 50.0000,GEAR_JERK 100.000,EXAX_IGN 0,CB {AUX_PT {ORI #CONSIDER,E1 #CONSIDER,E2 #CONSIDER,E3 #CONSIDER,E4 #CONSIDER,E5 #CONSIDER,E6 #CONSIDER},TARGET_PT {ORI #INTERPOLATE,E1 #INTERPOLATE,E2 #INTERPOLATE,E3 #INTERPOLATE,E4 #INTERPOLATE,E5 #INTERPOLATE,E6 #INTERPOLATE}}}
DECL E6POS XUS_TeachPick2_4={X 256.298584,Y -3.02997303,Z 6.21667910,A 90.8425293,B 0.983898640,C -179.492264,S 2,T 34,E1 0.0,E2 0.0,E3 0.0,E4 0.0,E5 0.0,E6 0.0}
DECL FDAT FUS_TeachPick2_4={TOOL_NO 1,BASE_NO 1,IPO_FRAME #BASE,POINT2[] " "}
DECL LDAT LCPDAT14={VEL 1.00000,ACC 60.0000,APO_DIST 500.000,APO_FAC 50.0000,AXIS_VEL 100.000,AXIS_ACC 60.0000,ORI_TYP #VAR,CIRC_TYP #BASE,JERK_FAC 50.0000,GEAR_JERK 100.000,EXAX_IGN 0,CB {AUX_PT {ORI #CONSIDER,E1 #CONSIDER,E2 #CONSIDER,E3 #CONSIDER,E4 #CONSIDER,E5 #CONSIDER,E6 #CONSIDER},TARGET_PT {ORI #INTERPOLATE,E1 #INTERPOLATE,E2 #INTERPOLATE,E3 #INTERPOLATE,E4 #INTERPOLATE,E5 #INTERPOLATE,E6 #INTERPOLATE}}}
DECL LDAT LCPDAT15={VEL 1.00000,ACC 60.0000,APO_DIST 500.000,APO_FAC 50.0000,AXIS_VEL 100.000,AXIS_ACC 60.0000,ORI_TYP #VAR,CIRC_TYP #BASE,JERK_FAC 50.0000,GEAR_JERK 100.000,EXAX_IGN 0,CB {AUX_PT {ORI #CONSIDER,E1 #CONSIDER,E2 #CONSIDER,E3 #CONSIDER,E4 #CONSIDER,E5 #CONSIDER,E6 #CONSIDER},TARGET_PT {ORI #INTERPOLATE,E1 #INTERPOLATE,E2 #INTERPOLATE,E3 #INTERPOLATE,E4 #INTERPOLATE,E5 #INTERPOLATE,E6 #INTERPOLATE}}}
DECL E6POS XUS_TeachPickstart={X 0.345544547,Y 180.631943,Z 82.0918274,A 90.0592346,B 1.36682498,C -179.299393,S 2,T 34,E1 0.0,E2 0.0,E3 0.0,E4 0.0,E5 0.0,E6 0.0}
DECL FDAT FUS_TeachPickstart={TOOL_NO 1,BASE_NO 1,IPO_FRAME #BASE,POINT2[] " "}
DECL PDAT PPDAT8={VEL 100.000,ACC 60.0000,APO_DIST 500.000,APO_MODE #CDIS,GEAR_JERK 100.000,EXAX_IGN 0}
DECL E6POS XDS_TeachPickStart={X 122.733109,Y 174.808395,Z 120.279678,A 88.9124,B 3.17389894,C 179.939789,S 2,T 10,E1 0.0,E2 0.0,E3 0.0,E4 0.0,E5 0.0,E6 0.0}
DECL FDAT FDS_TeachPickStart={TOOL_NO 2,BASE_NO 5,IPO_FRAME #BASE,POINT2[] " "}
DECL PDAT PPDAT9={VEL 100.000,ACC 60.0000,APO_DIST 500.000,APO_MODE #CDIS,GEAR_JERK 100.000,EXAX_IGN 0}
DECL E6POS XDS_TeachPick={X 4.31534386,Y 251.666153,Z -20.9911156,A 89.0877914,B 3.17406774,C 179.949509,S 2,T 10,E1 0.0,E2 0.0,E3 0.0,E4 0.0,E5 0.0,E6 0.0}
DECL FDAT FDS_TeachPick={TOOL_NO 2,BASE_NO 5,IPO_FRAME #BASE,POINT2[] " "}
DECL LDAT LCPDAT16={VEL 1.00000,ACC 60.0000,APO_DIST 500.000,APO_FAC 50.0000,AXIS_VEL 100.000,AXIS_ACC 60.0000,ORI_TYP #VAR,CIRC_TYP #BASE,JERK_FAC 50.0000,GEAR_JERK 100.000,EXAX_IGN 0,CB {AUX_PT {ORI #CONSIDER,E1 #CONSIDER,E2 #CONSIDER,E3 #CONSIDER,E4 #CONSIDER,E5 #CONSIDER,E6 #CONSIDER},TARGET_PT {ORI #INTERPOLATE,E1 #INTERPOLATE,E2 #INTERPOLATE,E3 #INTERPOLATE,E4 #INTERPOLATE,E5 #INTERPOLATE,E6 #INTERPOLATE}}}
DECL E6POS XDS_TeachPick1_2={X 55.0613289,Y 250.967255,Z -19.0239544,A 89.0877914,B 3.17406821,C 179.949509,S 2,T 10,E1 0.0,E2 0.0,E3 0.0,E4 0.0,E5 0.0,E6 0.0}
DECL FDAT FDS_TeachPick1_2={TOOL_NO 2,BASE_NO 5,IPO_FRAME #BASE,POINT2[] " "}
DECL LDAT LCPDAT17={VEL 1.00000,ACC 60.0000,APO_DIST 500.000,APO_FAC 50.0000,AXIS_VEL 100.000,AXIS_ACC 60.0000,ORI_TYP #VAR,CIRC_TYP #BASE,JERK_FAC 50.0000,GEAR_JERK 100.000,EXAX_IGN 0,CB {AUX_PT {ORI #CONSIDER,E1 #CONSIDER,E2 #CONSIDER,E3 #CONSIDER,E4 #CONSIDER,E5 #CONSIDER,E6 #CONSIDER},TARGET_PT {ORI #INTERPOLATE,E1 #INTERPOLATE,E2 #INTERPOLATE,E3 #INTERPOLATE,E4 #INTERPOLATE,E5 #INTERPOLATE,E6 #INTERPOLATE}}}
DECL E6POS XDS_TeachPick1_3={X 207.503403,Y 248.336212,Z -18.9673786,A 89.0863190,B 3.17473650,C 179.949142,S 2,T 10,E1 0.0,E2 0.0,E3 0.0,E4 0.0,E5 0.0,E6 0.0}
DECL FDAT FDS_TeachPick1_3={TOOL_NO 2,BASE_NO 5,IPO_FRAME #BASE,POINT2[] " "}
DECL LDAT LCPDAT18={VEL 1.00000,ACC 60.0000,APO_DIST 500.000,APO_FAC 50.0000,AXIS_VEL 100.000,AXIS_ACC 60.0000,ORI_TYP #VAR,CIRC_TYP #BASE,JERK_FAC 50.0000,GEAR_JERK 100.000,EXAX_IGN 0,CB {AUX_PT {ORI #CONSIDER,E1 #CONSIDER,E2 #CONSIDER,E3 #CONSIDER,E4 #CONSIDER,E5 #CONSIDER,E6 #CONSIDER},TARGET_PT {ORI #INTERPOLATE,E1 #INTERPOLATE,E2 #INTERPOLATE,E3 #INTERPOLATE,E4 #INTERPOLATE,E5 #INTERPOLATE,E6 #INTERPOLATE}}}
DECL PDAT PPDAT10={VEL 100.000,ACC 60.0000,APO_DIST 500.000,APO_MODE #CDIS,GEAR_JERK 100.000,EXAX_IGN 0}
DECL LDAT LCPDAT19={VEL 1.00000,ACC 60.0000,APO_DIST 500.000,APO_FAC 50.0000,AXIS_VEL 100.000,AXIS_ACC 60.0000,ORI_TYP #VAR,CIRC_TYP #BASE,JERK_FAC 50.0000,GEAR_JERK 100.000,EXAX_IGN 0,CB {AUX_PT {ORI #CONSIDER,E1 #CONSIDER,E2 #CONSIDER,E3 #CONSIDER,E4 #CONSIDER,E5 #CONSIDER,E6 #CONSIDER},TARGET_PT {ORI #INTERPOLATE,E1 #INTERPOLATE,E2 #INTERPOLATE,E3 #INTERPOLATE,E4 #INTERPOLATE,E5 #INTERPOLATE,E6 #INTERPOLATE}}}
DECL E6POS XDS_TeachPick1_4={X 258.334473,Y 247.107925,Z -19.4200420,A 89.0877914,B 3.17406821,C 179.949509,S 2,T 10,E1 0.0,E2 0.0,E3 0.0,E4 0.0,E5 0.0,E6 0.0}
DECL FDAT FDS_TeachPick1_4={TOOL_NO 2,BASE_NO 5,IPO_FRAME #BASE,POINT2[] " "}
DECL LDAT LCPDAT20={VEL 1.00000,ACC 60.0000,APO_DIST 500.000,APO_FAC 50.0000,AXIS_VEL 100.000,AXIS_ACC 60.0000,ORI_TYP #VAR,CIRC_TYP #BASE,JERK_FAC 50.0000,GEAR_JERK 100.000,EXAX_IGN 0,CB {AUX_PT {ORI #CONSIDER,E1 #CONSIDER,E2 #CONSIDER,E3 #CONSIDER,E4 #CONSIDER,E5 #CONSIDER,E6 #CONSIDER},TARGET_PT {ORI #INTERPOLATE,E1 #INTERPOLATE,E2 #INTERPOLATE,E3 #INTERPOLATE,E4 #INTERPOLATE,E5 #INTERPOLATE,E6 #INTERPOLATE}}}
DECL PDAT PPDAT12={VEL 100.000,ACC 60.0000,APO_DIST 500.000,APO_MODE #CDIS,GEAR_JERK 100.000,EXAX_IGN 0}
DECL LDAT LCPDAT21={VEL 1.00000,ACC 60.0000,APO_DIST 500.000,APO_FAC 50.0000,AXIS_VEL 100.000,AXIS_ACC 60.0000,ORI_TYP #VAR,CIRC_TYP #BASE,JERK_FAC 50.0000,GEAR_JERK 100.000,EXAX_IGN 0,CB {AUX_PT {ORI #CONSIDER,E1 #CONSIDER,E2 #CONSIDER,E3 #CONSIDER,E4 #CONSIDER,E5 #CONSIDER,E6 #CONSIDER},TARGET_PT {ORI #INTERPOLATE,E1 #INTERPOLATE,E2 #INTERPOLATE,E3 #INTERPOLATE,E4 #INTERPOLATE,E5 #INTERPOLATE,E6 #INTERPOLATE}}}
DECL E6POS XDS_TeachPick2_1={X 0.458416492,Y 66.8986893,Z -9.06041908,A 89.0877914,B 3.17424536,C 179.949493,S 2,T 10,E1 0.0,E2 0.0,E3 0.0,E4 0.0,E5 0.0,E6 0.0}
DECL FDAT FDS_TeachPick2_1={TOOL_NO 2,BASE_NO 5,IPO_FRAME #BASE,POINT2[] " "}
DECL LDAT LCPDAT22={VEL 1.00000,ACC 60.0000,APO_DIST 500.000,APO_FAC 50.0000,AXIS_VEL 100.000,AXIS_ACC 60.0000,ORI_TYP #VAR,CIRC_TYP #BASE,JERK_FAC 50.0000,GEAR_JERK 100.000,EXAX_IGN 0,CB {AUX_PT {ORI #CONSIDER,E1 #CONSIDER,E2 #CONSIDER,E3 #CONSIDER,E4 #CONSIDER,E5 #CONSIDER,E6 #CONSIDER},TARGET_PT {ORI #INTERPOLATE,E1 #INTERPOLATE,E2 #INTERPOLATE,E3 #INTERPOLATE,E4 #INTERPOLATE,E5 #INTERPOLATE,E6 #INTERPOLATE}}}
DECL E6POS XDS_TeachPick2_2={X 51.4475555,Y 66.5287476,Z -6.61884165,A 89.0877914,B 3.17424536,C 179.949493,S 2,T 10,E1 0.0,E2 0.0,E3 0.0,E4 0.0,E5 0.0,E6 0.0}
DECL FDAT FDS_TeachPick2_2={TOOL_NO 2,BASE_NO 5,IPO_FRAME #BASE,POINT2[] " "}
DECL LDAT LCPDAT23={VEL 1.00000,ACC 60.0000,APO_DIST 500.000,APO_FAC 50.0000,AXIS_VEL 100.000,AXIS_ACC 60.0000,ORI_TYP #VAR,CIRC_TYP #BASE,JERK_FAC 50.0000,GEAR_JERK 100.000,EXAX_IGN 0,CB {AUX_PT {ORI #CONSIDER,E1 #CONSIDER,E2 #CONSIDER,E3 #CONSIDER,E4 #CONSIDER,E5 #CONSIDER,E6 #CONSIDER},TARGET_PT {ORI #INTERPOLATE,E1 #INTERPOLATE,E2 #INTERPOLATE,E3 #INTERPOLATE,E4 #INTERPOLATE,E5 #INTERPOLATE,E6 #INTERPOLATE}}}
DECL E6POS XDS_TeachPick2_3={X 203.953934,Y 64.2239838,Z -9.19014263,A 89.0877914,B 3.17424536,C 179.949493,S 2,T 10,E1 0.0,E2 0.0,E3 0.0,E4 0.0,E5 0.0,E6 0.0}
DECL FDAT FDS_TeachPick2_3={TOOL_NO 2,BASE_NO 5,IPO_FRAME #BASE,POINT2[] " "}
DECL LDAT LCPDAT24={VEL 1.00000,ACC 60.0000,APO_DIST 500.000,APO_FAC 50.0000,AXIS_VEL 100.000,AXIS_ACC 60.0000,ORI_TYP #VAR,CIRC_TYP #BASE,JERK_FAC 50.0000,GEAR_JERK 100.000,EXAX_IGN 0,CB {AUX_PT {ORI #CONSIDER,E1 #CONSIDER,E2 #CONSIDER,E3 #CONSIDER,E4 #CONSIDER,E5 #CONSIDER,E6 #CONSIDER},TARGET_PT {ORI #INTERPOLATE,E1 #INTERPOLATE,E2 #INTERPOLATE,E3 #INTERPOLATE,E4 #INTERPOLATE,E5 #INTERPOLATE,E6 #INTERPOLATE}}}
DECL E6POS XDS_TeachPick2_4={X 254.851456,Y 63.3608284,Z -10.1410131,A 89.0877914,B 3.17424536,C 179.949493,S 2,T 10,E1 0.0,E2 0.0,E3 0.0,E4 0.0,E5 0.0,E6 0.0}
DECL FDAT FDS_TeachPick2_4={TOOL_NO 2,BASE_NO 5,IPO_FRAME #BASE,POINT2[] " "}
DECL LDAT LCPDAT25={VEL 1.00000,ACC 60.0000,APO_DIST 500.000,APO_FAC 50.0000,AXIS_VEL 100.000,AXIS_ACC 60.0000,ORI_TYP #VAR,CIRC_TYP #BASE,JERK_FAC 50.0000,GEAR_JERK 100.000,EXAX_IGN 0,CB {AUX_PT {ORI #CONSIDER,E1 #CONSIDER,E2 #CONSIDER,E3 #CONSIDER,E4 #CONSIDER,E5 #CONSIDER,E6 #CONSIDER},TARGET_PT {ORI #INTERPOLATE,E1 #INTERPOLATE,E2 #INTERPOLATE,E3 #INTERPOLATE,E4 #INTERPOLATE,E5 #INTERPOLATE,E6 #INTERPOLATE}}}
ENDDAT
